LIN {X 0,Y 196.128,Z 397.935,A -85,B 0,C 180,E1 -25531.035,E2 -25531.035} C_VEL
LIN {X 0,Y 198.391,Z 377.082,A -85,B 0,C 180,E1 -25531.639,E2 -25531.639} C_VEL
LIN {X 0,Y 200.245,Z 356.522,A -85,B 0,C 180,E1 -25532.183,E2 -25532.183} C_VEL
LIN {X 0,Y 201.46,Z 342.377,A -85,B 0,C 180,E1 -25532.591,E2 -25532.591} C_VEL
LIN {X 0,Y 197.272,Z 333.633,A -85,B 0,C 180,E1 -25535.814,E2 -25535.814} C_VEL
LIN {X 0,Y 193.686,Z 326.841,A -85,B 0,C 180,E1 -25539.002,E2 -25539.002} C_VEL
LIN {X 0,Y 190.138,Z 320.569,A -85,B 0,C 180,E1 -25542.8,E2 -25542.8} C_VEL
LIN {X 0,Y 187.785,Z 316.689,A -85,B 0,C 180,E1 -25545.92,E2 -25545.92} C_VEL
LIN {X 0,Y 185.741,Z 312.981,A -85,B 0,C 180,E1 -25549.508,E2 -25549.508} C_VEL
LIN {X 0,Y 183.942,Z 310.156,A -85,B 0,C 180,E1 -25554.291,E2 -25554.291} C_VEL
LIN {X 0,Y 183.571,Z 308.41,A -85,B 0,C 180,E1 -25556.708,E2 -25556.708} C_VEL
LIN {X 0,Y 183.342,Z 308.073,A -85,B 0,C 180,E1 -25560,E2 -25560} C_VEL
LIN {X 0,Y 183.573,Z 308.503,A -85,B 0,C 180,E1 -25563.017,E2 -25563.017} C_VEL
LIN {X 0,Y 185.059,Z 312.287,A -85,B 0,C 180,E1 -25568.737,E2 -25568.737} C_VEL
LIN {X 0,Y 185.908,Z 313.347,A -85,B 0,C 180,E1 -25570.493,E2 -25570.493} C_VEL
LIN {X 0,Y 188.57,Z 317.975,A -85,B 0,C 180,E1 -25574.846,E2 -25574.846} C_VEL
LIN {X 0,Y 191.002,Z 322.156,A -85,B 0,C 180,E1 -25577.864,E2 -25577.864} C_VEL
LIN {X 0,Y 194.086,Z 327.519,A -85,B 0,C 180,E1 -25581.021,E2 -25581.021} C_VEL
LIN {X 0,Y 196.464,Z 332.994,A -85,B 0,C 180,E1 -25583.242,E2 -25583.242} C_VEL
LIN {X 0,Y 199.811,Z 341.873,A -85,B 0,C 180,E1 -25586.082,E2 -25586.082} C_VEL
LIN {X 0,Y 201.242,Z 345.874,A -85,B 0,C 180,E1 -25587.202,E2 -25587.202} C_VEL
LIN {X 0,Y 196.159,Z 400.089,A -85,B 0,C 180,E1 -25588.654,E2 -25588.654} C_VEL
LIN {X 0,Y 193.398,Z 415.894,A -85,B 0,C 180,E1 -25589.293,E2 -25589.293} C_VEL
LIN {X 0,Y 189.564,Z 431.114,A -85,B 0,C 180,E1 -25590.2,E2 -25590.2} C_VEL
LIN {X 0,Y 185.029,Z 444.833,A -85,B 0,C 180,E1 -25591.284,E2 -25591.284} C_VEL
LIN {X 0,Y 179.626,Z 458.278,A -85,B 0,C 180,E1 -25592.735,E2 -25592.735} C_VEL
LIN {X 0,Y 173.796,Z 470.579,A -85,B 0,C 180,E1 -25594.481,E2 -25594.481} C_VEL
LIN {X 0,Y 166.767,Z 483.312,A -85,B 0,C 180,E1 -25596.804,E2 -25596.804} C_VEL
LIN {X 0,Y 159.457,Z 494.789,A -85,B 0,C 180,E1 -25599.531,E2 -25599.531} C_VEL
LIN {X 0,Y 152.65,Z 504.457,A -85,B 0,C 180,E1 -25602.556,E2 -25602.556} C_VEL
LIN {X 0,Y 146.078,Z 512.968,A -85,B 0,C 180,E1 -25605.958,E2 -25605.958} C_VEL
LIN {X 0,Y 139.091,Z 521.559,A -85,B 0,C 180,E1 -25610.53,E2 -25610.53} C_VEL
LIN {X 0,Y 132.199,Z 529.29,A -85,B 0,C 180,E1 -25616.069,E2 -25616.069} C_VEL
LIN {X 0,Y 127.359,Z 534.671,A -85,B 0,C 180,E1 -25621.352,E2 -25621.352} C_VEL
LIN {X 0,Y 124.98,Z 536.675,A -85,B 0,C 180,E1 -25623.643,E2 -25623.643} C_VEL
LIN {X 0,Y 119.742,Z 539.495,A -85,B 0,C 180,E1 -25627.37,E2 -25627.37} C_VEL
LIN {X 0,Y 115.773,Z 541.36,A -85,B 0,C 180,E1 -25630.607,E2 -25630.607} C_VEL
LIN {X 0,Y 113.779,Z 542.553,A -85,B 0,C 180,E1 -25633.329,E2 -25633.329} C_VEL
LIN {X 0,Y 113.428,Z 542.855,A -85,B 0,C 180,E1 -25634.29,E2 -25634.29} C_VEL
LIN {X 0,Y 112.457,Z 544.368,A -85,B 0,C 180,E1 -25639.194,E2 -25639.194} C_VEL
LIN {X 0,Y 112.095,Z 545.556,A -85,B 0,C 180,E1 -25646.406,E2 -25646.406} C_VEL
LIN {X 0,Y 112.248,Z 545.716,A -85,B 0,C 180,E1 -25650,E2 -25650} C_VEL
LIN {X 0,Y 112.127,Z 545.085,A -85,B 0,C 180,E1 -25657.201,E2 -25657.201} C_VEL
LIN {X 0,Y 113.102,Z 543.298,A -85,B 0,C 180,E1 -25664.392,E2 -25664.392} C_VEL
LIN {X 0,Y 115.541,Z 540.339,A -85,B 0,C 180,E1 -25671.405,E2 -25671.405} C_VEL
LIN {X 0,Y 119.379,Z 536.141,A -85,B 0,C 180,E1 -25678.097,E2 -25678.097} C_VEL
LIN {X 0,Y 124.755,Z 530.598,A -85,B 0,C 180,E1 -25684.286,E2 -25684.286} C_VEL
LIN {X 0,Y 131.504,Z 523.564,A -85,B 0,C 180,E1 -25689.889,E2 -25689.889} C_VEL
LIN {X 0,Y 138.144,Z 515.994,A -85,B 0,C 180,E1 -25694.427,E2 -25694.427} C_VEL
LIN {X 0,Y 145.607,Z 506.981,A -85,B 0,C 180,E1 -25698.428,E2 -25698.428} C_VEL
LIN {X 0,Y 153.787,Z 496.099,A -85,B 0,C 180,E1 -25702.027,E2 -25702.027} C_VEL
LIN {X 0,Y 161.311,Z 484.904,A -85,B 0,C 180,E1 -25704.774,E2 -25704.774} C_VEL
LIN {X 0,Y 168.603,Z 472.403,A -85,B 0,C 180,E1 -25707.128,E2 -25707.128} C_VEL
LIN {X 0,Y 175.176,Z 459.138,A -85,B 0,C 180,E1 -25709.041,E2 -25709.041} C_VEL
LIN {X 0,Y 180.723,Z 445.878,A -85,B 0,C 180,E1 -25710.471,E2 -25710.471} C_VEL
LIN {X 0,Y 185.34,Z 432.494,A -85,B 0,C 180,E1 -25711.551,E2 -25711.551} C_VEL
LIN {X 0,Y 189.296,Z 417.833,A -85,B 0,C 180,E1 -25712.422,E2 -25712.422} C_VEL
LIN {X 0,Y 192.258,Z 402.311,A -85,B 0,C 180,E1 -25713.067,E2 -25713.067} C_VEL
LIN {X 0,Y 194.771,Z 378.935,A -85,B 0,C 180,E1 -25713.717,E2 -25713.717} C_VEL
LIN {X 0,Y 197.573,Z 348.8,A -85,B 0,C 180,E1 -25714.503,E2 -25714.503} C_VEL
LIN {X 0,Y 194.226,Z 339.095,A -85,B 0,C 180,E1 -25717.53,E2 -25717.53} C_VEL
LIN {X 0,Y 192.008,Z 333.701,A -85,B 0,C 180,E1 -25719.727,E2 -25719.727} C_VEL
LIN {X 0,Y 188.543,Z 327.214,A -85,B 0,C 180,E1 -25723.586,E2 -25723.586} C_VEL
LIN {X 0,Y 186.245,Z 323.237,A -85,B 0,C 180,E1 -25726.776,E2 -25726.776} C_VEL
LIN {X 0,Y 184.286,Z 319.627,A -85,B 0,C 180,E1 -25730.396,E2 -25730.396} C_VEL
LIN {X 0,Y 182.581,Z 316.368,A -85,B 0,C 180,E1 -25735.585,E2 -25735.585} C_VEL
LIN {X 0,Y 182.365,Z 315.273,A -85,B 0,C 180,E1 -25737.239,E2 -25737.239} C_VEL
LIN {X 0,Y 182.148,Z 315.035,A -85,B 0,C 180,E1 -25740,E2 -25740} C_VEL
LIN {X 0,Y 182.427,Z 315.532,A -85,B 0,C 180,E1 -25743.728,E2 -25743.728} C_VEL
LIN {X 0,Y 183.832,Z 319.146,A -85,B 0,C 180,E1 -25749.074,E2 -25749.074} C_VEL
LIN {X 0,Y 184.588,Z 320.208,A -85,B 0,C 180,E1 -25750.697,E2 -25750.697} C_VEL
LIN {X 0,Y 186.924,Z 324.488,A -85,B 0,C 180,E1 -25754.702,E2 -25754.702} C_VEL
LIN {X 0,Y 189.274,Z 328.678,A -85,B 0,C 180,E1 -25757.764,E2 -25757.764} C_VEL
LIN {X 0,Y 191.987,Z 333.709,A -85,B 0,C 180,E1 -25760.701,E2 -25760.701} C_VEL
LIN {X 0,Y 195.196,Z 340.186,A -85,B 0,C 180,E1 -25763.683,E2 -25763.683} C_VEL
LIN {X 0,Y 197.771,Z 345.762,A -85,B 0,C 180,E1 -25765.81,E2 -25765.81} C_VEL
LIN {X 0,Y 193.113,Z 394.413,A -85,B 0,C 180,E1 -25767.114,E2 -25767.114} C_VEL
LIN {X 0,Y 190.393,Z 410.31,A -85,B 0,C 180,E1 -25767.78,E2 -25767.78} C_VEL
LIN {X 0,Y 186.718,Z 425.002,A -85,B 0,C 180,E1 -25768.663,E2 -25768.663} C_VEL
LIN {X 0,Y 182.252,Z 438.791,A -85,B 0,C 180,E1 -25769.816,E2 -25769.816} C_VEL
LIN {X 0,Y 177.003,Z 452.127,A -85,B 0,C 180,E1 -25771.323,E2 -25771.323} C_VEL
LIN {X 0,Y 171.009,Z 464.77,A -85,B 0,C 180,E1 -25773.14,E2 -25773.14} C_VEL
LIN {X 0,Y 164.504,Z 476.331,A -85,B 0,C 180,E1 -25775.21,E2 -25775.21} C_VEL
LIN {X 0,Y 157.683,Z 487.067,A -85,B 0,C 180,E1 -25777.711,E2 -25777.711} C_VEL
LIN {X 0,Y 150.546,Z 496.993,A -85,B 0,C 180,E1 -25780.66,E2 -25780.66} C_VEL
LIN {X 0,Y 143.003,Z 506.676,A -85,B 0,C 180,E1 -25784.553,E2 -25784.553} C_VEL
LIN {X 0,Y 135.891,Z 514.75,A -85,B 0,C 180,E1 -25788.747,E2 -25788.747} C_VEL
LIN {X 0,Y 129.57,Z 521.41,A -85,B 0,C 180,E1 -25793.37,E2 -25793.37} C_VEL
LIN {X 0,Y 123.476,Z 527.564,A -85,B 0,C 180,E1 -25799.186,E2 -25799.186} C_VEL
LIN {X 0,Y 118.71,Z 532.307,A -85,B 0,C 180,E1 -25805.518,E2 -25805.518} C_VEL
LIN {X 0,Y 115.253,Z 535.773,A -85,B 0,C 180,E1 -25812.249,E2 -25812.249} C_VEL
LIN {X 0,Y 113.198,Z 538.054,A -85,B 0,C 180,E1 -25819.266,E2 -25819.266} C_VEL
LIN {X 0,Y 112.353,Z 539.21,A -85,B 0,C 180,E1 -25826.414,E2 -25826.414} C_VEL
LIN {X 0,Y 112.335,Z 539.362,A -85,B 0,C 180,E1 -25830,E2 -25830} C_VEL
LIN {X 0,Y 112.624,Z 538.802,A -85,B 0,C 180,E1 -25837.169,E2 -25837.169} C_VEL
LIN {X 0,Y 114.05,Z 537.13,A -85,B 0,C 180,E1 -25844.269,E2 -25844.269} C_VEL
LIN {X 0,Y 116.718,Z 534.305,A -85,B 0,C 180,E1 -25851.178,E2 -25851.178} C_VEL
LIN {X 0,Y 120.946,Z 530.247,A -85,B 0,C 180,E1 -25857.701,E2 -25857.701} C_VEL
LIN {X 0,Y 126.368,Z 524.865,A -85,B 0,C 180,E1 -25863.789,E2 -25863.789} C_VEL
LIN {X 0,Y 133.011,Z 517.999,A -85,B 0,C 180,E1 -25869.349,E2 -25869.349} C_VEL
LIN {X 0,Y 140.769,Z 509.421,A -85,B 0,C 180,E1 -25874.342,E2 -25874.342} C_VEL
LIN {X 0,Y 147.586,Z 501.119,A -85,B 0,C 180,E1 -25878.012,E2 -25878.012} C_VEL
LIN {X 0,Y 155.159,Z 491.003,A -85,B 0,C 180,E1 -25881.382,E2 -25881.382} C_VEL
LIN {X 0,Y 162.498,Z 479.953,A -85,B 0,C 180,E1 -25884.185,E2 -25884.185} C_VEL
LIN {X 0,Y 169.582,Z 467.84,A -85,B 0,C 180,E1 -25886.514,E2 -25886.514} C_VEL
LIN {X 0,Y 175.733,Z 455.423,A -85,B 0,C 180,E1 -25888.398,E2 -25888.398} C_VEL
LIN {X 0,Y 180.809,Z 443.245,A -85,B 0,C 180,E1 -25889.863,E2 -25889.863} C_VEL
LIN {X 0,Y 185.929,Z 428.329,A -85,B 0,C 180,E1 -25891.217,E2 -25891.217} C_VEL
LIN {X 0,Y 189.927,Z 413.246,A -85,B 0,C 180,E1 -25892.202,E2 -25892.202} C_VEL
LIN {X 0,Y 192.784,Z 398.214,A -85,B 0,C 180,E1 -25892.874,E2 -25892.874} C_VEL
LIN {X 0,Y 195.151,Z 377.016,A -85,B 0,C 180,E1 -25893.474,E2 -25893.474} C_VEL
LIN {X 0,Y 196.842,Z 358.585,A -85,B 0,C 180,E1 -25893.969,E2 -25893.969} C_VEL
LIN {X 0,Y 197.973,Z 345.87,A -85,B 0,C 180,E1 -25894.332,E2 -25894.332} C_VEL
LIN {X 0,Y 194.145,Z 337.65,A -85,B 0,C 180,E1 -25897.59,E2 -25897.59} C_VEL
LIN {X 0,Y 190.481,Z 330.553,A -85,B 0,C 180,E1 -25901.27,E2 -25901.27} C_VEL
LIN {X 0,Y 188.099,Z 326.329,A -85,B 0,C 180,E1 -25904.144,E2 -25904.144} C_VEL
LIN {X 0,Y 186.4,Z 323.297,A -85,B 0,C 180,E1 -25906.619,E2 -25906.619} C_VEL
LIN {X 0,Y 184.406,Z 319.665,A -85,B 0,C 180,E1 -25910.402,E2 -25910.402} C_VEL
LIN {X 0,Y 182.733,Z 316.096,A -85,B 0,C 180,E1 -25916.141,E2 -25916.141} C_VEL
LIN {X 0,Y 182.63,Z 315.373,A -85,B 0,C 180,E1 -25917.243,E2 -25917.243} C_VEL
LIN {X 0,Y 182.477,Z 315.121,A -85,B 0,C 180,E1 -25920,E2 -25920} C_VEL
LIN {X 0,Y 182.67,Z 315.579,A -85,B 0,C 180,E1 -25922.825,E2 -25922.825} C_VEL
LIN {X 0,Y 184.076,Z 319.279,A -85,B 0,C 180,E1 -25928.508,E2 -25928.508} C_VEL
LIN {X 0,Y 184.77,Z 320.244,A -85,B 0,C 180,E1 -25930.028,E2 -25930.028} C_VEL
LIN {X 0,Y 187.212,Z 324.704,A -85,B 0,C 180,E1 -25934.262,E2 -25934.262} C_VEL
LIN {X 0,Y 189.498,Z 328.843,A -85,B 0,C 180,E1 -25937.259,E2 -25937.259} C_VEL
LIN {X 0,Y 192.256,Z 333.937,A -85,B 0,C 180,E1 -25940.251,E2 -25940.251} C_VEL
LIN {X 0,Y 194.505,Z 339.504,A -85,B 0,C 180,E1 -25942.49,E2 -25942.49} C_VEL
LIN {X 0,Y 197.731,Z 348.761,A -85,B 0,C 180,E1 -25945.407,E2 -25945.407} C_VEL
LIN {X 0,Y 197.495,Z 352.481,A -85,B 0,C 180,E1 -25945.57,E2 -25945.57} C_VEL
LIN {X 0,Y 192.822,Z 400.102,A -85,B 0,C 180,E1 -25946.807,E2 -25946.807} C_VEL
LIN {X 0,Y 190.035,Z 415.703,A -85,B 0,C 180,E1 -25947.432,E2 -25947.432} C_VEL
LIN {X 0,Y 186.098,Z 430.92,A -85,B 0,C 180,E1 -25948.312,E2 -25948.312} C_VEL
LIN {X 0,Y 181.442,Z 444.638,A -85,B 0,C 180,E1 -25949.367,E2 -25949.367} C_VEL
LIN {X 0,Y 175.887,Z 458.082,A -85,B 0,C 180,E1 -25950.788,E2 -25950.788} C_VEL
LIN {X 0,Y 169.464,Z 471.172,A -85,B 0,C 180,E1 -25952.624,E2 -25952.624} C_VEL
LIN {X 0,Y 161.953,Z 484.186,A -85,B 0,C 180,E1 -25955.008,E2 -25955.008} C_VEL
LIN {X 0,Y 153.794,Z 496.35,A -85,B 0,C 180,E1 -25957.977,E2 -25957.977} C_VEL
LIN {X 0,Y 145.615,Z 507.182,A -85,B 0,C 180,E1 -25961.576,E2 -25961.576} C_VEL
LIN {X 0,Y 138.219,Z 516.099,A -85,B 0,C 180,E1 -25965.541,E2 -25965.541} C_VEL
LIN {X 0,Y 131.509,Z 523.718,A -85,B 0,C 180,E1 -25970.113,E2 -25970.113} C_VEL
LIN {X 0,Y 124.778,Z 530.716,A -85,B 0,C 180,E1 -25975.721,E2 -25975.721} C_VEL
LIN {X 0,Y 119.282,Z 536.375,A -85,B 0,C 180,E1 -25982.102,E2 -25982.102} C_VEL
LIN {X 0,Y 115.57,Z 540.407,A -85,B 0,C 180,E1 -25988.601,E2 -25988.601} C_VEL
LIN {X 0,Y 113.428,Z 542.855,A -85,B 0,C 180,E1 -25994.29,E2 -25994.29} C_VEL
LIN {X 0,Y 112.204,Z 543.852,A -85,B 0,C 180,E1 -25997.178,E2 -25997.178} C_VEL
LIN {X 0,Y 109.003,Z 544.995,A -85,B 0,C 180,E1 -26001.986,E2 -26001.986} C_VEL
LIN {X 0,Y 105.6,Z 545.541,A -85,B 0,C 180,E1 -26008.126,E2 -26008.126} C_VEL
LIN {X 0,Y 105.138,Z 545.503,A -85,B 0,C 180,E1 -26010.282,E2 -26010.282} C_VEL
LIN {X 0,Y 105.053,Z 544.883,A -85,B 0,C 180,E1 -26017.689,E2 -26017.689} C_VEL
LIN {X 0,Y 106.184,Z 543.095,A -85,B 0,C 180,E1 -26025.352,E2 -26025.352} C_VEL
LIN {X 0,Y 108.884,Z 540.135,A -85,B 0,C 180,E1 -26032.785,E2 -26032.785} C_VEL
LIN {X 0,Y 113.108,Z 535.937,A -85,B 0,C 180,E1 -26039.806,E2 -26039.806} C_VEL
LIN {X 0,Y 118.895,Z 530.394,A -85,B 0,C 180,E1 -26046.235,E2 -26046.235} C_VEL
LIN {X 0,Y 126.06,Z 523.358,A -85,B 0,C 180,E1 -26051.99,E2 -26051.99} C_VEL
LIN {X 0,Y 133.554,Z 515.296,A -85,B 0,C 180,E1 -26056.836,E2 -26056.836} C_VEL
LIN {X 0,Y 140.964,Z 506.777,A -85,B 0,C 180,E1 -26060.602,E2 -26060.602} C_VEL
LIN {X 0,Y 149.493,Z 495.894,A -85,B 0,C 180,E1 -26064.188,E2 -26064.188} C_VEL
LIN {X 0,Y 157.313,Z 484.7,A -85,B 0,C 180,E1 -26066.892,E2 -26066.892} C_VEL
LIN {X 0,Y 165.105,Z 471.735,A -85,B 0,C 180,E1 -26069.283,E2 -26069.283} C_VEL
LIN {X 0,Y 171.628,Z 458.933,A -85,B 0,C 180,E1 -26071.077,E2 -26071.077} C_VEL
LIN {X 0,Y 177.327,Z 445.672,A -85,B 0,C 180,E1 -26072.47,E2 -26072.47} C_VEL
LIN {X 0,Y 182.069,Z 432.286,A -85,B 0,C 180,E1 -26073.513,E2 -26073.513} C_VEL
LIN {X 0,Y 186.12,Z 417.623,A -85,B 0,C 180,E1 -26074.358,E2 -26074.358} C_VEL
LIN {X 0,Y 189.102,Z 402.418,A -85,B 0,C 180,E1 -26074.97,E2 -26074.97} C_VEL
LIN {X 0,Y 191.639,Z 379.78,A -85,B 0,C 180,E1 -26075.587,E2 -26075.587} C_VEL
LIN {X 0,Y 194.302,Z 351.818,A -85,B 0,C 180,E1 -26076.313,E2 -26076.313} C_VEL
LIN {X 0,Y 191.403,Z 343.066,A -85,B 0,C 180,E1 -26079.234,E2 -26079.234} C_VEL
LIN {X 0,Y 189.685,Z 339.028,A -85,B 0,C 180,E1 -26081.083,E2 -26081.083} C_VEL
LIN {X 0,Y 186.8,Z 333.397,A -85,B 0,C 180,E1 -26084.591,E2 -26084.591} C_VEL
LIN {X 0,Y 184.86,Z 329.819,A -85,B 0,C 180,E1 -26087.513,E2 -26087.513} C_VEL
LIN {X 0,Y 183.131,Z 326.461,A -85,B 0,C 180,E1 -26090.961,E2 -26090.961} C_VEL
LIN {X 0,Y 181.541,Z 322.805,A -85,B 0,C 180,E1 -26096.671,E2 -26096.671} C_VEL
LIN {X 0,Y 181.425,Z 322.252,A -85,B 0,C 180,E1 -26097.78,E2 -26097.78} C_VEL
LIN {X 0,Y 181.437,Z 322.287,A -85,B 0,C 180,E1 -26102.776,E2 -26102.776} C_VEL
LIN {X 0,Y 183.089,Z 326.414,A -85,B 0,C 180,E1 -26109.389,E2 -26109.389} C_VEL
LIN {X 0,Y 185.397,Z 330.78,A -85,B 0,C 180,E1 -26113.802,E2 -26113.802} C_VEL
LIN {X 0,Y 187.834,Z 335.446,A -85,B 0,C 180,E1 -26117.207,E2 -26117.207} C_VEL
LIN {X 0,Y 190.678,Z 341.118,A -85,B 0,C 180,E1 -26120.426,E2 -26120.426} C_VEL
LIN {X 0,Y 193.81,Z 347.891,A -85,B 0,C 180,E1 -26123.441,E2 -26123.441} C_VEL
LIN {X 0,Y 194.453,Z 349.345,A -85,B 0,C 180,E1 -26124.009,E2 -26124.009} C_VEL
LIN {X 0,Y 189.897,Z 395.315,A -85,B 0,C 180,E1 -26125.238,E2 -26125.238} C_VEL
LIN {X 0,Y 187.193,Z 410.521,A -85,B 0,C 180,E1 -26125.859,E2 -26125.859} C_VEL
LIN {X 0,Y 183.429,Z 425.211,A -85,B 0,C 180,E1 -26126.723,E2 -26126.723} C_VEL
LIN {X 0,Y 178.824,Z 438.999,A -85,B 0,C 180,E1 -26127.84,E2 -26127.84} C_VEL
LIN {X 0,Y 173.211,Z 452.802,A -85,B 0,C 180,E1 -26129.373,E2 -26129.373} C_VEL
LIN {X 0,Y 166.561,Z 466.262,A -85,B 0,C 180,E1 -26131.304,E2 -26131.304} C_VEL
LIN {X 0,Y 159.211,Z 478.664,A -85,B 0,C 180,E1 -26133.574,E2 -26133.574} C_VEL
LIN {X 0,Y 152.16,Z 489.045,A -85,B 0,C 180,E1 -26136.072,E2 -26136.072} C_VEL
LIN {X 0,Y 144.086,Z 499.542,A -85,B 0,C 180,E1 -26139.353,E2 -26139.353} C_VEL
LIN {X 0,Y 136.978,Z 508.102,A -85,B 0,C 180,E1 -26143.02,E2 -26143.02} C_VEL
LIN {X 0,Y 129.609,Z 515.954,A -85,B 0,C 180,E1 -26147.329,E2 -26147.329} C_VEL
LIN {X 0,Y 122.173,Z 523.278,A -85,B 0,C 180,E1 -26152.843,E2 -26152.843} C_VEL
LIN {X 0,Y 115.975,Z 529.079,A -85,B 0,C 180,E1 -26158.997,E2 -26158.997} C_VEL
LIN {X 0,Y 112.273,Z 532.509,A -85,B 0,C 180,E1 -26164.013,E2 -26164.013} C_VEL
LIN {X 0,Y 108.478,Z 535.975,A -85,B 0,C 180,E1 -26171.099,E2 -26171.099} C_VEL
LIN {X 0,Y 106.212,Z 538.256,A -85,B 0,C 180,E1 -26178.55,E2 -26178.55} C_VEL
LIN {X 0,Y 105.265,Z 539.411,A -85,B 0,C 180,E1 -26186.172,E2 -26186.172} C_VEL
LIN {X 0,Y 105.237,Z 539.563,A -85,B 0,C 180,E1 -26190,E2 -26190} C_VEL
LIN {X 0,Y 105.592,Z 539.003,A -85,B 0,C 180,E1 -26197.649,E2 -26197.649} C_VEL
LIN {X 0,Y 107.157,Z 537.331,A -85,B 0,C 180,E1 -26205.209,E2 -26205.209} C_VEL
LIN {X 0,Y 110.094,Z 534.506,A -85,B 0,C 180,E1 -26212.52,E2 -26212.52} C_VEL
LIN {X 0,Y 114.654,Z 530.449,A -85,B 0,C 180,E1 -26219.365,E2 -26219.365} C_VEL
LIN {X 0,Y 120.496,Z 525.066,A -85,B 0,C 180,E1 -26225.679,E2 -26225.679} C_VEL
LIN {X 0,Y 127.58,Z 518.199,A -85,B 0,C 180,E1 -26231.378,E2 -26231.378} C_VEL
LIN {X 0,Y 134.663,Z 510.816,A -85,B 0,C 180,E1 -26235.856,E2 -26235.856} C_VEL
LIN {X 0,Y 141.344,Z 503.199,A -85,B 0,C 180,E1 -26239.355,E2 -26239.355} C_VEL
LIN {X 0,Y 147.146,Z 496.054,A -85,B 0,C 180,E1 -26242.004,E2 -26242.004} C_VEL
LIN {X 0,Y 154.657,Z 485.912,A -85,B 0,C 180,E1 -26244.879,E2 -26244.879} C_VEL
LIN {X 0,Y 161.081,Z 475.963,A -85,B 0,C 180,E1 -26247.125,E2 -26247.125} C_VEL
LIN {X 0,Y 168.494,Z 462.994,A -85,B 0,C 180,E1 -26249.346,E2 -26249.346} C_VEL
LIN {X 0,Y 174.472,Z 450.327,A -85,B 0,C 180,E1 -26251.093,E2 -26251.093} C_VEL
LIN {X 0,Y 180.152,Z 435.959,A -85,B 0,C 180,E1 -26252.559,E2 -26252.559} C_VEL
LIN {X 0,Y 184.773,Z 421.22,A -85,B 0,C 180,E1 -26253.663,E2 -26253.663} C_VEL
LIN {X 0,Y 188.18,Z 406.625,A -85,B 0,C 180,E1 -26254.466,E2 -26254.466} C_VEL
LIN {X 0,Y 190.714,Z 390.557,A -85,B 0,C 180,E1 -26255.032,E2 -26255.032} C_VEL
LIN {X 0,Y 192.711,Z 370.089,A -85,B 0,C 180,E1 -26255.588,E2 -26255.588} C_VEL
LIN {X 0,Y 194.695,Z 349.528,A -85,B 0,C 180,E1 -26256.106,E2 -26256.106} C_VEL
LIN {X 0,Y 191.57,Z 342.573,A -85,B 0,C 180,E1 -26259.041,E2 -26259.041} C_VEL
LIN {X 0,Y 188.427,Z 336.273,A -85,B 0,C 180,E1 -26262.499,E2 -26262.499} C_VEL
LIN {X 0,Y 186.624,Z 332.876,A -85,B 0,C 180,E1 -26264.86,E2 -26264.86} C_VEL
LIN {X 0,Y 185.088,Z 330.002,A -85,B 0,C 180,E1 -26267.249,E2 -26267.249} C_VEL
LIN {X 0,Y 183.297,Z 326.501,A -85,B 0,C 180,E1 -26270.9,E2 -26270.9} C_VEL
LIN {X 0,Y 181.792,Z 322.923,A -85,B 0,C 180,E1 -26276.675,E2 -26276.675} C_VEL
LIN {X 0,Y 181.704,Z 322.347,A -85,B 0,C 180,E1 -26277.783,E2 -26277.783} C_VEL
LIN {X 0,Y 181.645,Z 322.261,A -85,B 0,C 180,E1 -26281.108,E2 -26281.108} C_VEL
LIN {X 0,Y 181.767,Z 322.671,A -85,B 0,C 180,E1 -26282.631,E2 -26282.631} C_VEL
LIN {X 0,Y 183.095,Z 326.274,A -85,B 0,C 180,E1 -26288.276,E2 -26288.276} C_VEL
LIN {X 0,Y 183.692,Z 327.201,A -85,B 0,C 180,E1 -26289.659,E2 -26289.659} C_VEL
LIN {X 0,Y 185.874,Z 331.433,A -85,B 0,C 180,E1 -26293.669,E2 -26293.669} C_VEL
LIN {X 0,Y 187.954,Z 335.392,A -85,B 0,C 180,E1 -26296.565,E2 -26296.565} C_VEL
LIN {X 0,Y 190.76,Z 340.985,A -85,B 0,C 180,E1 -26299.784,E2 -26299.784} C_VEL
LIN {X 0,Y 193.285,Z 348.192,A -85,B 0,C 180,E1 -26302.444,E2 -26302.444} C_VEL
LIN {X 0,Y 194.524,Z 352.047,A -85,B 0,C 180,E1 -26303.652,E2 -26303.652} C_VEL
LIN {X 0,Y 189.706,Z 400.09,A -85,B 0,C 180,E1 -26304.904,E2 -26304.904} C_VEL
LIN {X 0,Y 186.859,Z 415.511,A -85,B 0,C 180,E1 -26305.492,E2 -26305.492} C_VEL
LIN {X 0,Y 182.841,Z 430.726,A -85,B 0,C 180,E1 -26306.355,E2 -26306.355} C_VEL
LIN {X 0,Y 178.066,Z 444.442,A -85,B 0,C 180,E1 -26307.375,E2 -26307.375} C_VEL
LIN {X 0,Y 172.357,Z 457.886,A -85,B 0,C 180,E1 -26308.758,E2 -26308.758} C_VEL
LIN {X 0,Y 166.014,Z 470.454,A -85,B 0,C 180,E1 -26310.474,E2 -26310.474} C_VEL
LIN {X 0,Y 158.644,Z 482.916,A -85,B 0,C 180,E1 -26312.681,E2 -26312.681} C_VEL
LIN {X 0,Y 150.754,Z 494.39,A -85,B 0,C 180,E1 -26315.332,E2 -26315.332} C_VEL
LIN {X 0,Y 143.355,Z 504.057,A -85,B 0,C 180,E1 -26318.336,E2 -26318.336} C_VEL
LIN {X 0,Y 135.263,Z 513.558,A -85,B 0,C 180,E1 -26322.236,E2 -26322.236} C_VEL
LIN {X 0,Y 128.011,Z 521.485,A -85,B 0,C 180,E1 -26326.666,E2 -26326.666} C_VEL
LIN {X 0,Y 120.555,Z 528.886,A -85,B 0,C 180,E1 -26332.258,E2 -26332.258} C_VEL
LIN {X 0,Y 114.462,Z 534.769,A -85,B 0,C 180,E1 -26338.541,E2 -26338.541} C_VEL
LIN {X 0,Y 110.885,Z 538.277,A -85,B 0,C 180,E1 -26343.663,E2 -26343.663} C_VEL
LIN {X 0,Y 107.318,Z 541.822,A -85,B 0,C 180,E1 -26350.887,E2 -26350.887} C_VEL
LIN {X 0,Y 105.463,Z 544.167,A -85,B 0,C 180,E1 -26358.468,E2 -26358.468} C_VEL
LIN {X 0,Y 105.005,Z 545.355,A -85,B 0,C 180,E1 -26366.162,E2 -26366.162} C_VEL
LIN {X 0,Y 105.138,Z 545.503,A -85,B 0,C 180,E1 -26370.282,E2 -26370.282} C_VEL
LIN {X 0,Y 104.271,Z 545.349,A -85,B 0,C 180,E1 -26373.475,E2 -26373.475} C_VEL
LIN {X 0,Y 101.537,Z 544.676,A -85,B 0,C 180,E1 -26378.775,E2 -26378.775} C_VEL
LIN {X 0,Y 99.684,Z 543.768,A -85,B 0,C 180,E1 -26383.182,E2 -26383.182} C_VEL
LIN {X 0,Y 99.396,Z 542.856,A -85,B 0,C 180,E1 -26386.568,E2 -26386.568} C_VEL
LIN {X 0,Y 99.626,Z 542.484,A -85,B 0,C 180,E1 -26387.685,E2 -26387.685} C_VEL
LIN {X 0,Y 102.3,Z 539.932,A -85,B 0,C 180,E1 -26394.343,E2 -26394.343} C_VEL
LIN {X 0,Y 106.942,Z 535.733,A -85,B 0,C 180,E1 -26401.717,E2 -26401.717} C_VEL
LIN {X 0,Y 113.178,Z 530.189,A -85,B 0,C 180,E1 -26408.386,E2 -26408.386} C_VEL
LIN {X 0,Y 120.824,Z 523.154,A -85,B 0,C 180,E1 -26414.266,E2 -26414.266} C_VEL
LIN {X 0,Y 128.167,Z 515.711,A -85,B 0,C 180,E1 -26418.852,E2 -26418.852} C_VEL
LIN {X 0,Y 136.53,Z 506.572,A -85,B 0,C 180,E1 -26422.926,E2 -26422.926} C_VEL
LIN {X 0,Y 145.416,Z 495.689,A -85,B 0,C 180,E1 -26426.478,E2 -26426.478} C_VEL
LIN {X 0,Y 153.539,Z 484.495,A -85,B 0,C 180,E1 -26429.119,E2 -26429.119} C_VEL
LIN {X 0,Y 161.037,Z 472.448,A -85,B 0,C 180,E1 -26431.311,E2 -26431.311} C_VEL
LIN {X 0,Y 168.293,Z 458.726,A -85,B 0,C 180,E1 -26433.203,E2 -26433.203} C_VEL
LIN {X 0,Y 174.154,Z 445.465,A -85,B 0,C 180,E1 -26434.545,E2 -26434.545} C_VEL
LIN {X 0,Y 179.013,Z 432.078,A -85,B 0,C 180,E1 -26435.549,E2 -26435.549} C_VEL
LIN {X 0,Y 183.163,Z 417.413,A -85,B 0,C 180,E1 -26436.358,E2 -26436.358} C_VEL
LIN {X 0,Y 186.243,Z 401.971,A -85,B 0,C 180,E1 -26436.96,E2 -26436.96} C_VEL
LIN {X 0,Y 188.911,Z 378.6,A -85,B 0,C 180,E1 -26437.572,E2 -26437.572} C_VEL
LIN {X 0,Y 191.202,Z 354.974,A -85,B 0,C 180,E1 -26438.193,E2 -26438.193} C_VEL
LIN {X 0,Y 189.01,Z 347.982,A -85,B 0,C 180,E1 -26440.661,E2 -26440.661} C_VEL
LIN {X 0,Y 187.355,Z 344.152,A -85,B 0,C 180,E1 -26442.607,E2 -26442.607} C_VEL
LIN {X 0,Y 185.056,Z 339.435,A -85,B 0,C 180,E1 -26445.709,E2 -26445.709} C_VEL
LIN {X 0,Y 183.544,Z 336.474,A -85,B 0,C 180,E1 -26448.193,E2 -26448.193} C_VEL
LIN {X 0,Y 182.054,Z 333.339,A -85,B 0,C 180,E1 -26451.397,E2 -26451.397} C_VEL
LIN {X 0,Y 180.621,Z 329.781,A -85,B 0,C 180,E1 -26457.003,E2 -26457.003} C_VEL
LIN {X 0,Y 180.56,Z 329.306,A -85,B 0,C 180,E1 -26457.77,E2 -26457.77} C_VEL
LIN {X 0,Y 180.507,Z 329.298,A -85,B 0,C 180,E1 -26462.232,E2 -26462.232} C_VEL
LIN {X 0,Y 180.645,Z 329.965,A -85,B 0,C 180,E1 -26463.695,E2 -26463.695} C_VEL
LIN {X 0,Y 181.985,Z 333.268,A -85,B 0,C 180,E1 -26468.887,E2 -26468.887} C_VEL
LIN {X 0,Y 184.035,Z 337.372,A -85,B 0,C 180,E1 -26473.103,E2 -26473.103} C_VEL
LIN {X 0,Y 186.261,Z 341.887,A -85,B 0,C 180,E1 -26476.439,E2 -26476.439} C_VEL
LIN {X 0,Y 189.169,Z 348.042,A -85,B 0,C 180,E1 -26479.924,E2 -26479.924} C_VEL
LIN {X 0,Y 191.366,Z 353.104,A -85,B 0,C 180,E1 -26482.189,E2 -26482.189} C_VEL
LIN {X 0,Y 186.918,Z 395.964,A -85,B 0,C 180,E1 -26483.29,E2 -26483.29} C_VEL
LIN {X 0,Y 184.028,Z 411.498,A -85,B 0,C 180,E1 -26483.915,E2 -26483.915} C_VEL
LIN {X 0,Y 179.989,Z 426.568,A -85,B 0,C 180,E1 -26484.795,E2 -26484.795} C_VEL
LIN {X 0,Y 174.908,Z 441.061,A -85,B 0,C 180,E1 -26485.969,E2 -26485.969} C_VEL
LIN {X 0,Y 168.893,Z 455.011,A -85,B 0,C 180,E1 -26487.532,E2 -26487.532} C_VEL
LIN {X 0,Y 162.283,Z 467.704,A -85,B 0,C 180,E1 -26489.363,E2 -26489.363} C_VEL
LIN {X 0,Y 154.717,Z 479.902,A -85,B 0,C 180,E1 -26491.603,E2 -26491.603} C_VEL
LIN {X 0,Y 146.771,Z 491.014,A -85,B 0,C 180,E1 -26494.312,E2 -26494.312} C_VEL
LIN {X 0,Y 138.234,Z 501.537,A -85,B 0,C 180,E1 -26497.774,E2 -26497.774} C_VEL
LIN {X 0,Y 131.057,Z 509.529,A -85,B 0,C 180,E1 -26501.345,E2 -26501.345} C_VEL
LIN {X 0,Y 123.425,Z 517.157,A -85,B 0,C 180,E1 -26505.772,E2 -26505.772} C_VEL
LIN {X 0,Y 116.562,Z 523.481,A -85,B 0,C 180,E1 -26510.723,E2 -26510.723} C_VEL
LIN {X 0,Y 109.918,Z 529.282,A -85,B 0,C 180,E1 -26517.08,E2 -26517.08} C_VEL
LIN {X 0,Y 105.908,Z 532.711,A -85,B 0,C 180,E1 -26522.322,E2 -26522.322} C_VEL
LIN {X 0,Y 101.76,Z 536.178,A -85,B 0,C 180,E1 -26529.799,E2 -26529.799} C_VEL
LIN {X 0,Y 99.257,Z 538.457,A -85,B 0,C 180,E1 -26537.736,E2 -26537.736} C_VEL
LIN {X 0,Y 98.189,Z 539.612,A -85,B 0,C 180,E1 -26545.896,E2 -26545.896} C_VEL
LIN {X 0,Y 98.151,Z 539.763,A -85,B 0,C 180,E1 -26550,E2 -26550} C_VEL
LIN {X 0,Y 98.553,Z 539.203,A -85,B 0,C 180,E1 -26558.199,E2 -26558.199} C_VEL
LIN {X 0,Y 100.306,Z 537.532,A -85,B 0,C 180,E1 -26566.275,E2 -26566.275} C_VEL
LIN {X 0,Y 103.54,Z 534.707,A -85,B 0,C 180,E1 -26574.032,E2 -26574.032} C_VEL
LIN {X 0,Y 108.475,Z 530.65,A -85,B 0,C 180,E1 -26581.218,E2 -26581.218} C_VEL
LIN {X 0,Y 114.773,Z 525.266,A -85,B 0,C 180,E1 -26587.758,E2 -26587.758} C_VEL
LIN {X 0,Y 122.32,Z 518.399,A -85,B 0,C 180,E1 -26593.587,E2 -26593.587} C_VEL
LIN {X 0,Y 129.812,Z 511.016,A -85,B 0,C 180,E1 -26598.108,E2 -26598.108} C_VEL
LIN {X 0,Y 137.574,Z 502.496,A -85,B 0,C 180,E1 -26602.012,E2 -26602.012} C_VEL
LIN {X 0,Y 145.405,Z 493.02,A -85,B 0,C 180,E1 -26605.251,E2 -26605.251} C_VEL
LIN {X 0,Y 153.266,Z 482.292,A -85,B 0,C 180,E1 -26608.027,E2 -26608.027} C_VEL
LIN {X 0,Y 160.775,Z 470.574,A -85,B 0,C 180,E1 -26610.317,E2 -26610.317} C_VEL
LIN {X 0,Y 167.736,Z 457.801,A -85,B 0,C 180,E1 -26612.251,E2 -26612.251} C_VEL
LIN {X 0,Y 173.407,Z 445.396,A -85,B 0,C 180,E1 -26613.725,E2 -26613.725} C_VEL
LIN {X 0,Y 178.447,Z 432.097,A -85,B 0,C 180,E1 -26614.933,E2 -26614.933} C_VEL
LIN {X 0,Y 182.823,Z 417.431,A -85,B 0,C 180,E1 -26615.918,E2 -26615.918} C_VEL
LIN {X 0,Y 186.146,Z 402.287,A -85,B 0,C 180,E1 -26616.622,E2 -26616.622} C_VEL
LIN {X 0,Y 188.375,Z 386.071,A -85,B 0,C 180,E1 -26617.109,E2 -26617.109} C_VEL
LIN {X 0,Y 191.596,Z 353.22,A -85,B 0,C 180,E1 -26617.946,E2 -26617.946} C_VEL
LIN {X 0,Y 188.628,Z 346.504,A -85,B 0,C 180,E1 -26621.079,E2 -26621.079} C_VEL
LIN {X 0,Y 185.733,Z 340.396,A -85,B 0,C 180,E1 -26624.786,E2 -26624.786} C_VEL
LIN {X 0,Y 183.817,Z 336.711,A -85,B 0,C 180,E1 -26627.861,E2 -26627.861} C_VEL
LIN {X 0,Y 182.2,Z 333.363,A -85,B 0,C 180,E1 -26631.404,E2 -26631.404} C_VEL
LIN {X 0,Y 180.867,Z 329.751,A -85,B 0,C 180,E1 -26637.216,E2 -26637.216} C_VEL
LIN {X 0,Y 180.759,Z 329.298,A -85,B 0,C 180,E1 -26638.886,E2 -26638.886} C_VEL
LIN {X 0,Y 180.851,Z 329.5,A -85,B 0,C 180,E1 -26642.088,E2 -26642.088} C_VEL
LIN {X 0,Y 182.118,Z 333.265,A -85,B 0,C 180,E1 -26648.041,E2 -26648.041} C_VEL
LIN {X 0,Y 182.612,Z 334.197,A -85,B 0,C 180,E1 -26649.274,E2 -26649.274} C_VEL
LIN {X 0,Y 184.478,Z 337.976,A -85,B 0,C 180,E1 -26652.933,E2 -26652.933} C_VEL
LIN {X 0,Y 186.573,Z 342.194,A -85,B 0,C 180,E1 -26656.038,E2 -26656.038} C_VEL
LIN {X 0,Y 188.873,Z 347.147,A -85,B 0,C 180,E1 -26658.86,E2 -26658.86} C_VEL
LIN {X 0,Y 191.117,Z 354.155,A -85,B 0,C 180,E1 -26661.434,E2 -26661.434} C_VEL
LIN {X 0,Y 191.475,Z 355.303,A -85,B 0,C 180,E1 -26661.816,E2 -26661.816} C_VEL
LIN {X 0,Y 186.823,Z 399.988,A -85,B 0,C 180,E1 -26662.939,E2 -26662.939} C_VEL
LIN {X 0,Y 183.905,Z 415.319,A -85,B 0,C 180,E1 -26663.488,E2 -26663.488} C_VEL
LIN {X 0,Y 179.801,Z 430.532,A -85,B 0,C 180,E1 -26664.327,E2 -26664.327} C_VEL
LIN {X 0,Y 174.915,Z 444.247,A -85,B 0,C 180,E1 -26665.309,E2 -26665.309} C_VEL
LIN {X 0,Y 169.037,Z 457.689,A -85,B 0,C 180,E1 -26666.635,E2 -26666.635} C_VEL
LIN {X 0,Y 162.102,Z 471.002,A -85,B 0,C 180,E1 -26668.414,E2 -26668.414} C_VEL
LIN {X 0,Y 154.228,Z 483.79,A -85,B 0,C 180,E1 -26670.673,E2 -26670.673} C_VEL
LIN {X 0,Y 145.424,Z 495.951,A -85,B 0,C 180,E1 -26673.526,E2 -26673.526} C_VEL
LIN {X 0,Y 136.54,Z 506.782,A -85,B 0,C 180,E1 -26677.079,E2 -26677.079} C_VEL
LIN {X 0,Y 128.246,Z 515.822,A -85,B 0,C 180,E1 -26681.118,E2 -26681.118} C_VEL
LIN {X 0,Y 120.832,Z 523.315,A -85,B 0,C 180,E1 -26685.738,E2 -26685.738} C_VEL
LIN {X 0,Y 113.198,Z 530.312,A -85,B 0,C 180,E1 -26691.622,E2 -26691.622} C_VEL
LIN {X 0,Y 106.992,Z 535.825,A -85,B 0,C 180,E1 -26698.299,E2 -26698.299} C_VEL
LIN {X 0,Y 102.347,Z 540.002,A -85,B 0,C 180,E1 -26705.67,E2 -26705.67} C_VEL
LIN {X 0,Y 99.299,Z 542.939,A -85,B 0,C 180,E1 -26713.555,E2 -26713.555} C_VEL
LIN {X 0,Y 98.005,Z 544.702,A -85,B 0,C 180,E1 -26721.754,E2 -26721.754} C_VEL
LIN {X 0,Y 98.066,Z 545.313,A -85,B 0,C 180,E1 -26730.056,E2 -26730.056} C_VEL
LIN {X 0,Y 98.004,Z 544.682,A -85,B 0,C 180,E1 -26738.246,E2 -26738.246} C_VEL
LIN {X 0,Y 99.285,Z 542.891,A -85,B 0,C 180,E1 -26746.448,E2 -26746.448} C_VEL
LIN {X 0,Y 99.626,Z 542.484,A -85,B 0,C 180,E1 -26747.685,E2 -26747.685} C_VEL
LIN {X 0,Y 100.081,Z 541.4,A -85,B 0,C 180,E1 -26751.002,E2 -26751.002} C_VEL
LIN {X 0,Y 99.719,Z 539.205,A -85,B 0,C 180,E1 -26756.555,E2 -26756.555} C_VEL
LIN {X 0,Y 99.925,Z 537.139,A -85,B 0,C 180,E1 -26760.968,E2 -26760.968} C_VEL
LIN {X 0,Y 101.204,Z 535.356,A -85,B 0,C 180,E1 -26764.1,E2 -26764.1} C_VEL
LIN {X 0,Y 101.943,Z 534.69,A -85,B 0,C 180,E1 -26765.066,E2 -26765.066} C_VEL
LIN {X 0,Y 109.567,Z 528.356,A -85,B 0,C 180,E1 -26772.337,E2 -26772.337} C_VEL
LIN {X 0,Y 117.928,Z 520.915,A -85,B 0,C 180,E1 -26778.153,E2 -26778.153} C_VEL
LIN {X 0,Y 126.047,Z 512.959,A -85,B 0,C 180,E1 -26782.61,E2 -26782.61} C_VEL
LIN {X 0,Y 134.938,Z 503.421,A -85,B 0,C 180,E1 -26786.44,E2 -26786.44} C_VEL
LIN {X 0,Y 142.959,Z 493.706,A -85,B 0,C 180,E1 -26789.35,E2 -26789.35} C_VEL
LIN {X 0,Y 151.426,Z 482.183,A -85,B 0,C 180,E1 -26791.862,E2 -26791.862} C_VEL
LIN {X 0,Y 159.311,Z 469.484,A -85,B 0,C 180,E1 -26794.004,E2 -26794.004} C_VEL
LIN {X 0,Y 165.945,Z 456.976,A -85,B 0,C 180,E1 -26795.579,E2 -26795.579} C_VEL
LIN {X 0,Y 171.951,Z 443.407,A -85,B 0,C 180,E1 -26796.868,E2 -26796.868} C_VEL
LIN {X 0,Y 177.324,Z 428.321,A -85,B 0,C 180,E1 -26797.882,E2 -26797.882} C_VEL
LIN {X 0,Y 181.355,Z 413.384,A -85,B 0,C 180,E1 -26798.588,E2 -26798.588} C_VEL
LIN {X 0,Y 184.098,Z 398.526,A -85,B 0,C 180,E1 -26799.101,E2 -26799.101} C_VEL
LIN {X 0,Y 188.314,Z 358.219,A -85,B 0,C 180,E1 -26800.121,E2 -26800.121} C_VEL
LIN {X 0,Y 186.58,Z 352.49,A -85,B 0,C 180,E1 -26802.321,E2 -26802.321} C_VEL
LIN {X 0,Y 184.054,Z 346.782,A -85,B 0,C 180,E1 -26805.793,E2 -26805.793} C_VEL
LIN {X 0,Y 182.256,Z 343.115,A -85,B 0,C 180,E1 -26808.884,E2 -26808.884} C_VEL
LIN {X 0,Y 180.962,Z 340.176,A -85,B 0,C 180,E1 -26811.907,E2 -26811.907} C_VEL
LIN {X 0,Y 179.698,Z 336.66,A -85,B 0,C 180,E1 -26817.478,E2 -26817.478} C_VEL
LIN {X 0,Y 179.553,Z 336.173,A -85,B 0,C 180,E1 -26820,E2 -26820} C_VEL
LIN {X 0,Y 179.699,Z 336.623,A -85,B 0,C 180,E1 -26822.943,E2 -26822.943} C_VEL
LIN {X 0,Y 180.869,Z 340.088,A -85,B 0,C 180,E1 -26828.308,E2 -26828.308} C_VEL
LIN {X 0,Y 182.64,Z 343.832,A -85,B 0,C 180,E1 -26832.279,E2 -26832.279} C_VEL
LIN {X 0,Y 184.96,Z 348.821,A -85,B 0,C 180,E1 -26835.991,E2 -26835.991} C_VEL
LIN {X 0,Y 187.778,Z 355.306,A -85,B 0,C 180,E1 -26839.543,E2 -26839.543} C_VEL
LIN {X 0,Y 188.444,Z 356.904,A -85,B 0,C 180,E1 -26840.287,E2 -26840.287} C_VEL
LIN {X 0,Y 184.339,Z 395.516,A -85,B 0,C 180,E1 -26841.244,E2 -26841.244} C_VEL
LIN {X 0,Y 181.46,Z 410.943,A -85,B 0,C 180,E1 -26841.83,E2 -26841.83} C_VEL
LIN {X 0,Y 177.501,Z 425.628,A -85,B 0,C 180,E1 -26842.629,E2 -26842.629} C_VEL
LIN {X 0,Y 172.652,Z 439.413,A -85,B 0,C 180,E1 -26843.671,E2 -26843.671} C_VEL
LIN {X 0,Y 166.789,Z 452.997,A -85,B 0,C 180,E1 -26845.079,E2 -26845.079} C_VEL
LIN {X 0,Y 159.649,Z 466.672,A -85,B 0,C 180,E1 -26846.948,E2 -26846.948} C_VEL
LIN {X 0,Y 151.806,Z 479.073,A -85,B 0,C 180,E1 -26849.095,E2 -26849.095} C_VEL
LIN {X 0,Y 144.254,Z 489.453,A -85,B 0,C 180,E1 -26851.507,E2 -26851.507} C_VEL
LIN {X 0,Y 136.286,Z 499.082,A -85,B 0,C 180,E1 -26854.405,E2 -26854.405} C_VEL
LIN {X 0,Y 127.709,Z 508.508,A -85,B 0,C 180,E1 -26858.355,E2 -26858.355} C_VEL
LIN {X 0,Y 119.519,Z 516.361,A -85,B 0,C 180,E1 -26862.692,E2 -26862.692} C_VEL
LIN {X 0,Y 111.144,Z 523.684,A -85,B 0,C 180,E1 -26868.399,E2 -26868.399} C_VEL
LIN {X 0,Y 104.003,Z 529.485,A -85,B 0,C 180,E1 -26874.944,E2 -26874.944} C_VEL
LIN {X 0,Y 99.637,Z 532.914,A -85,B 0,C 180,E1 -26880.413,E2 -26880.413} C_VEL
LIN {X 0,Y 95.11,Z 536.38,A -85,B 0,C 180,E1 -26888.318,E2 -26888.318} C_VEL
LIN {X 0,Y 92.311,Z 538.659,A -85,B 0,C 180,E1 -26896.797,E2 -26896.797} C_VEL
LIN {X 0,Y 91.106,Z 539.813,A -85,B 0,C 180,E1 -26905.576,E2 -26905.576} C_VEL
LIN {X 0,Y 91.056,Z 539.964,A -85,B 0,C 180,E1 -26910,E2 -26910} C_VEL
LIN {X 0,Y 91.541,Z 539.404,A -85,B 0,C 180,E1 -26918.832,E2 -26918.832} C_VEL
LIN {X 0,Y 93.475,Z 537.734,A -85,B 0,C 180,E1 -26927.502,E2 -26927.502} C_VEL
LIN {X 0,Y 97.067,Z 534.908,A -85,B 0,C 180,E1 -26935.748,E2 -26935.748} C_VEL
LIN {X 0,Y 102.429,Z 530.851,A -85,B 0,C 180,E1 -26943.291,E2 -26943.291} C_VEL
LIN {X 0,Y 109.221,Z 525.467,A -85,B 0,C 180,E1 -26950.049,E2 -26950.049} C_VEL
LIN {X 0,Y 117.258,Z 518.599,A -85,B 0,C 180,E1 -26955.99,E2 -26955.99} C_VEL
LIN {X 0,Y 125.183,Z 511.215,A -85,B 0,C 180,E1 -26960.528,E2 -26960.528} C_VEL
LIN {X 0,Y 132.878,Z 503.152,A -85,B 0,C 180,E1 -26964.243,E2 -26964.243} C_VEL
LIN {X 0,Y 141.464,Z 493.219,A -85,B 0,C 180,E1 -26967.624,E2 -26967.624} C_VEL
LIN {X 0,Y 148.262,Z 484.433,A -85,B 0,C 180,E1 -26969.892,E2 -26969.892} C_VEL
LIN {X 0,Y 155.953,Z 473.109,A -85,B 0,C 180,E1 -26972.175,E2 -26972.175} C_VEL
LIN {X 0,Y 163.125,Z 460.801,A -85,B 0,C 180,E1 -26974.072,E2 -26974.072} C_VEL
LIN {X 0,Y 169.657,Z 447.336,A -85,B 0,C 180,E1 -26975.689,E2 -26975.689} C_VEL
LIN {X 0,Y 175.196,Z 433.37,A -85,B 0,C 180,E1 -26976.943,E2 -26976.943} C_VEL
LIN {X 0,Y 179.664,Z 419.01,A -85,B 0,C 180,E1 -26977.906,E2 -26977.906} C_VEL
LIN {X 0,Y 183.186,Z 403.876,A -85,B 0,C 180,E1 -26978.596,E2 -26978.596} C_VEL
LIN {X 0,Y 185.517,Z 388.296,A -85,B 0,C 180,E1 -26979.068,E2 -26979.068} C_VEL
LIN {X 0,Y 188.672,Z 356.981,A -85,B 0,C 180,E1 -26979.861,E2 -26979.861} C_VEL
LIN {X 0,Y 185.835,Z 350.455,A -85,B 0,C 180,E1 -26983.275,E2 -26983.275} C_VEL
LIN {X 0,Y 183.711,Z 345.82,A -85,B 0,C 180,E1 -26986.42,E2 -26986.42} C_VEL
LIN {X 0,Y 182.358,Z 343.042,A -85,B 0,C 180,E1 -26988.889,E2 -26988.889} C_VEL
LIN {X 0,Y 181.144,Z 340.253,A -85,B 0,C 180,E1 -26991.845,E2 -26991.845} C_VEL
LIN {X 0,Y 179.924,Z 336.411,A -85,B 0,C 180,E1 -26998.321,E2 -26998.321} C_VEL
LIN {X 0,Y 179.954,Z 336.423,A -85,B 0,C 180,E1 -27001.678,E2 -27001.678} C_VEL
LIN {X 0,Y 180.89,Z 339.906,A -85,B 0,C 180,E1 -27007.101,E2 -27007.101} C_VEL
LIN {X 0,Y 181.451,Z 340.897,A -85,B 0,C 180,E1 -27008.632,E2 -27008.632} C_VEL
LIN {X 0,Y 183.186,Z 344.697,A -85,B 0,C 180,E1 -27012.322,E2 -27012.322} C_VEL
LIN {X 0,Y 184.999,Z 348.576,A -85,B 0,C 180,E1 -27015.21,E2 -27015.21} C_VEL
LIN {X 0,Y 187.038,Z 353.298,A -85,B 0,C 180,E1 -27017.917,E2 -27017.917} C_VEL
LIN {X 0,Y 188.567,Z 358.445,A -85,B 0,C 180,E1 -27019.858,E2 -27019.858} C_VEL
LIN {X 0,Y 184.29,Z 399.07,A -85,B 0,C 180,E1 -27020.881,E2 -27020.881} C_VEL
LIN {X 0,Y 181.189,Z 415.128,A -85,B 0,C 180,E1 -27021.425,E2 -27021.425} C_VEL
LIN {X 0,Y 176.999,Z 430.339,A -85,B 0,C 180,E1 -27022.236,E2 -27022.236} C_VEL
LIN {X 0,Y 171.996,Z 444.052,A -85,B 0,C 180,E1 -27023.167,E2 -27023.167} C_VEL
LIN {X 0,Y 165.96,Z 457.492,A -85,B 0,C 180,E1 -27024.432,E2 -27024.432} C_VEL
LIN {X 0,Y 159.064,Z 470.398,A -85,B 0,C 180,E1 -27026.095,E2 -27026.095} C_VEL
LIN {X 0,Y 151.423,Z 482.519,A -85,B 0,C 180,E1 -27028.136,E2 -27028.136} C_VEL
LIN {X 0,Y 142.971,Z 493.992,A -85,B 0,C 180,E1 -27030.658,E2 -27030.658} C_VEL
LIN {X 0,Y 134.962,Z 503.657,A -85,B 0,C 180,E1 -27033.575,E2 -27033.575} C_VEL
LIN {X 0,Y 126.077,Z 513.156,A -85,B 0,C 180,E1 -27037.408,E2 -27037.408} C_VEL
LIN {X 0,Y 117.944,Z 521.08,A -85,B 0,C 180,E1 -27041.856,E2 -27041.856} C_VEL
LIN {X 0,Y 109.568,Z 528.483,A -85,B 0,C 180,E1 -27047.664,E2 -27047.664} C_VEL
LIN {X 0,Y 102.498,Z 534.365,A -85,B 0,C 180,E1 -27054.352,E2 -27054.352} C_VEL
LIN {X 0,Y 98.206,Z 537.872,A -85,B 0,C 180,E1 -27059.938,E2 -27059.938} C_VEL
LIN {X 0,Y 93.929,Z 541.419,A -85,B 0,C 180,E1 -27068.031,E2 -27068.031} C_VEL
LIN {X 0,Y 91.501,Z 543.763,A -85,B 0,C 180,E1 -27076.678,E2 -27076.678} C_VEL
LIN {X 0,Y 90.807,Z 544.952,A -85,B 0,C 180,E1 -27085.561,E2 -27085.561} C_VEL
LIN {X 0,Y 90.969,Z 545.114,A -85,B 0,C 180,E1 -27090,E2 -27090} C_VEL
LIN {X 0,Y 90.95,Z 544.48,A -85,B 0,C 180,E1 -27098.89,E2 -27098.89} C_VEL
LIN {X 0,Y 92.642,Z 542.465,A -85,B 0,C 180,E1 -27108.431,E2 -27108.431} C_VEL
LIN {X 0,Y 95.801,Z 539.728,A -85,B 0,C 180,E1 -27116.114,E2 -27116.114} C_VEL
LIN {X 0,Y 100.912,Z 535.529,A -85,B 0,C 180,E1 -27123.859,E2 -27123.859} C_VEL
LIN {X 0,Y 101.943,Z 534.69,A -85,B 0,C 180,E1 -27125.066,E2 -27125.066} C_VEL
LIN {X 0,Y 103.937,Z 532.683,A -85,B 0,C 180,E1 -27127.948,E2 -27127.948} C_VEL
LIN {X 0,Y 106.137,Z 529.112,A -85,B 0,C 180,E1 -27132.844,E2 -27132.844} C_VEL
LIN {X 0,Y 108.849,Z 525.054,A -85,B 0,C 180,E1 -27137.451,E2 -27137.451} C_VEL
LIN {X 0,Y 111.529,Z 522.266,A -85,B 0,C 180,E1 -27139.78,E2 -27139.78} C_VEL
LIN {X 0,Y 120.565,Z 513.993,A -85,B 0,C 180,E1 -27144.693,E2 -27144.693} C_VEL
LIN {X 0,Y 129.757,Z 504.709,A -85,B 0,C 180,E1 -27148.544,E2 -27148.544} C_VEL
LIN {X 0,Y 138.043,Z 495.28,A -85,B 0,C 180,E1 -27151.427,E2 -27151.427} C_VEL
LIN {X 0,Y 147.463,Z 483.05,A -85,B 0,C 180,E1 -27154.099,E2 -27154.099} C_VEL
LIN {X 0,Y 155.575,Z 470.575,A -85,B 0,C 180,E1 -27156.172,E2 -27156.172} C_VEL
LIN {X 0,Y 162.37,Z 458.314,A -85,B 0,C 180,E1 -27157.694,E2 -27157.694} C_VEL
LIN {X 0,Y 168.524,Z 445.051,A -85,B 0,C 180,E1 -27158.922,E2 -27158.922} C_VEL
LIN {X 0,Y 173.997,Z 430.532,A -85,B 0,C 180,E1 -27159.898,E2 -27159.898} C_VEL
LIN {X 0,Y 178.323,Z 415.465,A -85,B 0,C 180,E1 -27160.63,E2 -27160.63} C_VEL
LIN {X 0,Y 181.418,Z 400.017,A -85,B 0,C 180,E1 -27161.142,E2 -27161.142} C_VEL
LIN {X 0,Y 185.4,Z 364.29,A -85,B 0,C 180,E1 -27161.996,E2 -27161.996} C_VEL
LIN {X 0,Y 185.636,Z 361.498,A -85,B 0,C 180,E1 -27162.114,E2 -27162.114} C_VEL
LIN {X 0,Y 184.458,Z 357.728,A -85,B 0,C 180,E1 -27163.769,E2 -27163.769} C_VEL
LIN {X 0,Y 182.237,Z 352.531,A -85,B 0,C 180,E1 -27167.188,E2 -27167.188} C_VEL
LIN {X 0,Y 180.9,Z 349.537,A -85,B 0,C 180,E1 -27169.79,E2 -27169.79} C_VEL
LIN {X 0,Y 179.881,Z 347.038,A -85,B 0,C 180,E1 -27172.423,E2 -27172.423} C_VEL
LIN {X 0,Y 178.758,Z 343.413,A -85,B 0,C 180,E1 -27178.347,E2 -27178.347} C_VEL
LIN {X 0,Y 178.697,Z 343.31,A -85,B 0,C 180,E1 -27181.127,E2 -27181.127} C_VEL
LIN {X 0,Y 178.802,Z 343.773,A -85,B 0,C 180,E1 -27182.816,E2 -27182.816} C_VEL
LIN {X 0,Y 180.136,Z 347.701,A -85,B 0,C 180,E1 -27188.766,E2 -27188.766} C_VEL
LIN {X 0,Y 181.774,Z 351.52,A -85,B 0,C 180,E1 -27192.424,E2 -27192.424} C_VEL
LIN {X 0,Y 183.752,Z 356.044,A -85,B 0,C 180,E1 -27195.672,E2 -27195.672} C_VEL
LIN {X 0,Y 185.71,Z 360.853,A -85,B 0,C 180,E1 -27198.321,E2 -27198.321} C_VEL
LIN {X 0,Y 181.785,Z 396.347,A -85,B 0,C 180,E1 -27199.179,E2 -27199.179} C_VEL
LIN {X 0,Y 178.755,Z 411.919,A -85,B 0,C 180,E1 -27199.76,E2 -27199.76} C_VEL
LIN {X 0,Y 174.516,Z 426.984,A -85,B 0,C 180,E1 -27200.562,E2 -27200.562} C_VEL
LIN {X 0,Y 169.169,Z 441.474,A -85,B 0,C 180,E1 -27201.638,E2 -27201.638} C_VEL
LIN {X 0,Y 163.011,Z 455.059,A -85,B 0,C 180,E1 -27203.056,E2 -27203.056} C_VEL
LIN {X 0,Y 155.818,Z 468.113,A -85,B 0,C 180,E1 -27204.811,E2 -27204.811} C_VEL
LIN {X 0,Y 147.772,Z 480.31,A -85,B 0,C 180,E1 -27206.91,E2 -27206.91} C_VEL
LIN {X 0,Y 139.256,Z 491.422,A -85,B 0,C 180,E1 -27209.477,E2 -27209.477} C_VEL
LIN {X 0,Y 130.199,Z 501.676,A -85,B 0,C 180,E1 -27212.67,E2 -27212.67} C_VEL
LIN {X 0,Y 122.136,Z 509.935,A -85,B 0,C 180,E1 -27216.334,E2 -27216.334} C_VEL
LIN {X 0,Y 113.639,Z 517.564,A -85,B 0,C 180,E1 -27220.748,E2 -27220.748} C_VEL
LIN {X 0,Y 105.922,Z 523.887,A -85,B 0,C 180,E1 -27225.84,E2 -27225.84} C_VEL
LIN {X 0,Y 98.248,Z 529.688,A -85,B 0,C 180,E1 -27232.554,E2 -27232.554} C_VEL
LIN {X 0,Y 93.497,Z 533.117,A -85,B 0,C 180,E1 -27238.253,E2 -27238.253} C_VEL
LIN {X 0,Y 88.518,Z 536.582,A -85,B 0,C 180,E1 -27246.611,E2 -27246.611} C_VEL
LIN {X 0,Y 85.405,Z 538.861,A -85,B 0,C 180,E1 -27255.708,E2 -27255.708} C_VEL
LIN {X 0,Y 84.05,Z 540.013,A -85,B 0,C 180,E1 -27265.204,E2 -27265.204} C_VEL
LIN {X 0,Y 83.956,Z 540.165,A -85,B 0,C 180,E1 -27270,E2 -27270} C_VEL
LIN {X 0,Y 84.513,Z 539.605,A -85,B 0,C 180,E1 -27279.573,E2 -27279.573} C_VEL
LIN {X 0,Y 86.703,Z 537.935,A -85,B 0,C 180,E1 -27288.919,E2 -27288.919} C_VEL
LIN {X 0,Y 90.693,Z 535.11,A -85,B 0,C 180,E1 -27297.706,E2 -27297.706} C_VEL
LIN {X 0,Y 96.539,Z 531.052,A -85,B 0,C 180,E1 -27305.618,E2 -27305.618} C_VEL
LIN {X 0,Y 103.86,Z 525.667,A -85,B 0,C 180,E1 -27312.583,E2 -27312.583} C_VEL
LIN {X 0,Y 112.41,Z 518.8,A -85,B 0,C 180,E1 -27318.611,E2 -27318.611} C_VEL
LIN {X 0,Y 120.79,Z 511.414,A -85,B 0,C 180,E1 -27323.131,E2 -27323.131} C_VEL
LIN {X 0,Y 129.398,Z 502.729,A -85,B 0,C 180,E1 -27327.103,E2 -27327.103} C_VEL
LIN {X 0,Y 137.792,Z 493.417,A -85,B 0,C 180,E1 -27330.118,E2 -27330.118} C_VEL
LIN {X 0,Y 146.234,Z 482.688,A -85,B 0,C 180,E1 -27332.759,E2 -27332.759} C_VEL
LIN {X 0,Y 154.233,Z 470.968,A -85,B 0,C 180,E1 -27334.908,E2 -27334.908} C_VEL
LIN {X 0,Y 160.891,Z 459.584,A -85,B 0,C 180,E1 -27336.534,E2 -27336.534} C_VEL
LIN {X 0,Y 166.861,Z 447.532,A -85,B 0,C 180,E1 -27337.909,E2 -27337.909} C_VEL
LIN {X 0,Y 172.545,Z 433.564,A -85,B 0,C 180,E1 -27339.108,E2 -27339.108} C_VEL
LIN {X 0,Y 177.121,Z 419.202,A -85,B 0,C 180,E1 -27340.031,E2 -27340.031} C_VEL
LIN {X 0,Y 180.848,Z 403.449,A -85,B 0,C 180,E1 -27340.713,E2 -27340.713} C_VEL
LIN {X 0,Y 183.272,Z 386.934,A -85,B 0,C 180,E1 -27341.183,E2 -27341.183} C_VEL
LIN {X 0,Y 185.945,Z 360.962,A -85,B 0,C 180,E1 -27341.826,E2 -27341.826} C_VEL
LIN {X 0,Y 183.552,Z 355.161,A -85,B 0,C 180,E1 -27345.143,E2 -27345.143} C_VEL
LIN {X 0,Y 181.546,Z 350.485,A -85,B 0,C 180,E1 -27348.698,E2 -27348.698} C_VEL
LIN {X 0,Y 180.05,Z 347.071,A -85,B 0,C 180,E1 -27352.43,E2 -27352.43} C_VEL
LIN {X 0,Y 179.056,Z 343.479,A -85,B 0,C 180,E1 -27358.313,E2 -27358.313} C_VEL
LIN {X 0,Y 179.054,Z 343.365,A -85,B 0,C 180,E1 -27361.124,E2 -27361.124} C_VEL
LIN {X 0,Y 180.358,Z 347.739,A -85,B 0,C 180,E1 -27368.12,E2 -27368.12} C_VEL
LIN {X 0,Y 181.971,Z 351.519,A -85,B 0,C 180,E1 -27371.804,E2 -27371.804} C_VEL
LIN {X 0,Y 183.986,Z 356.147,A -85,B 0,C 180,E1 -27375.154,E2 -27375.154} C_VEL
LIN {X 0,Y 185.282,Z 359.595,A -85,B 0,C 180,E1 -27377.003,E2 -27377.003} C_VEL
LIN {X 0,Y 185.911,Z 361.874,A -85,B 0,C 180,E1 -27377.9,E2 -27377.9} C_VEL
LIN {X 0,Y 181.882,Z 398.885,A -85,B 0,C 180,E1 -27378.793,E2 -27378.793} C_VEL
LIN {X 0,Y 178.718,Z 414.936,A -85,B 0,C 180,E1 -27379.306,E2 -27379.306} C_VEL
LIN {X 0,Y 174.437,Z 430.145,A -85,B 0,C 180,E1 -27380.078,E2 -27380.078} C_VEL
LIN {X 0,Y 169.319,Z 443.857,A -85,B 0,C 180,E1 -27380.95,E2 -27380.95} C_VEL
LIN {X 0,Y 163.149,Z 457.296,A -85,B 0,C 180,E1 -27382.159,E2 -27382.159} C_VEL
LIN {X 0,Y 155.604,Z 470.988,A -85,B 0,C 180,E1 -27383.853,E2 -27383.853} C_VEL
LIN {X 0,Y 147.461,Z 483.392,A -85,B 0,C 180,E1 -27385.9,E2 -27385.9} C_VEL
LIN {X 0,Y 138.054,Z 495.552,A -85,B 0,C 180,E1 -27388.582,E2 -27388.582} C_VEL
LIN {X 0,Y 128.437,Z 506.382,A -85,B 0,C 180,E1 -27391.991,E2 -27391.991} C_VEL
LIN {X 0,Y 119.302,Z 515.431,A -85,B 0,C 180,E1 -27395.934,E2 -27395.934} C_VEL
LIN {X 0,Y 111.015,Z 522.912,A -85,B 0,C 180,E1 -27400.565,E2 -27400.565} C_VEL
LIN {X 0,Y 102.345,Z 529.909,A -85,B 0,C 180,E1 -27406.632,E2 -27406.632} C_VEL
LIN {X 0,Y 95.076,Z 535.42,A -85,B 0,C 180,E1 -27413.748,E2 -27413.748} C_VEL
LIN {X 0,Y 89.457,Z 539.597,A -85,B 0,C 180,E1 -27421.877,E2 -27421.877} C_VEL
LIN {X 0,Y 85.648,Z 542.534,A -85,B 0,C 180,E1 -27430.839,E2 -27430.839} C_VEL
LIN {X 0,Y 83.9,Z 544.299,A -85,B 0,C 180,E1 -27440.356,E2 -27440.356} C_VEL
LIN {X 0,Y 83.875,Z 544.913,A -85,B 0,C 180,E1 -27450,E2 -27450} C_VEL
LIN {X 0,Y 83.728,Z 544.744,A -85,B 0,C 180,E1 -27454.815,E2 -27454.815} C_VEL
LIN {X 0,Y 84.552,Z 543.526,A -85,B 0,C 180,E1 -27464.439,E2 -27464.439} C_VEL
LIN {X 0,Y 87.29,Z 541.154,A -85,B 0,C 180,E1 -27473.738,E2 -27473.738} C_VEL
LIN {X 0,Y 91.986,Z 537.584,A -85,B 0,C 180,E1 -27482.331,E2 -27482.331} C_VEL
LIN {X 0,Y 98.501,Z 532.73,A -85,B 0,C 180,E1 -27489.951,E2 -27489.951} C_VEL
LIN {X 0,Y 106.503,Z 526.46,A -85,B 0,C 180,E1 -27496.54,E2 -27496.54} C_VEL
LIN {X 0,Y 111.529,Z 522.266,A -85,B 0,C 180,E1 -27499.78,E2 -27499.78} C_VEL
LIN {X 0,Y 114.327,Z 519.404,A -85,B 0,C 180,E1 -27501.974,E2 -27501.974} C_VEL
LIN {X 0,Y 121.028,Z 510.294,A -85,B 0,C 180,E1 -27508.716,E2 -27508.716} C_VEL
LIN {X 0,Y 123.966,Z 506.827,A -85,B 0,C 180,E1 -27510.472,E2 -27510.472} C_VEL
LIN {X 0,Y 125.115,Z 505.6,A -85,B 0,C 180,E1 -27510.94,E2 -27510.94} C_VEL
LIN {X 0,Y 134.768,Z 495.075,A -85,B 0,C 180,E1 -27514.099,E2 -27514.099} C_VEL
LIN {X 0,Y 144.487,Z 482.844,A -85,B 0,C 180,E1 -27516.647,E2 -27516.647} C_VEL
LIN {X 0,Y 152.83,Z 470.369,A -85,B 0,C 180,E1 -27518.621,E2 -27518.621} C_VEL
LIN {X 0,Y 159.8,Z 458.108,A -85,B 0,C 180,E1 -27520.06,E2 -27520.06} C_VEL
LIN {X 0,Y 166.096,Z 444.844,A -85,B 0,C 180,E1 -27521.214,E2 -27521.214} C_VEL
LIN {X 0,Y 171.685,Z 430.324,A -85,B 0,C 180,E1 -27522.124,E2 -27522.124} C_VEL
LIN {X 0,Y 176.098,Z 415.254,A -85,B 0,C 180,E1 -27522.807,E2 -27522.807} C_VEL
LIN {X 0,Y 179.166,Z 400.269,A -85,B 0,C 180,E1 -27523.279,E2 -27523.279} C_VEL
LIN {X 0,Y 182.532,Z 371.518,A -85,B 0,C 180,E1 -27523.94,E2 -27523.94} C_VEL
LIN {X 0,Y 183.201,Z 365.147,A -85,B 0,C 180,E1 -27524.097,E2 -27524.097} C_VEL
LIN {X 0,Y 181.364,Z 360.239,A -85,B 0,C 180,E1 -27527.055,E2 -27527.055} C_VEL
LIN {X 0,Y 179.75,Z 356.322,A -85,B 0,C 180,E1 -27530.329,E2 -27530.329} C_VEL
LIN {X 0,Y 178.792,Z 353.861,A -85,B 0,C 180,E1 -27533.015,E2 -27533.015} C_VEL
LIN {X 0,Y 177.891,Z 350.475,A -85,B 0,C 180,E1 -27538.339,E2 -27538.339} C_VEL
LIN {X 0,Y 177.861,Z 350.426,A -85,B 0,C 180,E1 -27541.698,E2 -27541.698} C_VEL
LIN {X 0,Y 179.029,Z 354.473,A -85,B 0,C 180,E1 -27548.181,E2 -27548.181} C_VEL
LIN {X 0,Y 180.428,Z 357.995,A -85,B 0,C 180,E1 -27551.616,E2 -27551.616} C_VEL
LIN {X 0,Y 182.184,Z 362.319,A -85,B 0,C 180,E1 -27554.772,E2 -27554.772} C_VEL
LIN {X 0,Y 183.165,Z 364.956,A -85,B 0,C 180,E1 -27556.281,E2 -27556.281} C_VEL
LIN {X 0,Y 179.551,Z 396.739,A -85,B 0,C 180,E1 -27557.048,E2 -27557.048} C_VEL
LIN {X 0,Y 176.484,Z 412.129,A -85,B 0,C 180,E1 -27557.594,E2 -27557.594} C_VEL
LIN {X 0,Y 172.156,Z 427.191,A -85,B 0,C 180,E1 -27558.355,E2 -27558.355} C_VEL
LIN {X 0,Y 166.689,Z 441.68,A -85,B 0,C 180,E1 -27559.376,E2 -27559.376} C_VEL
LIN {X 0,Y 160.675,Z 454.657,A -85,B 0,C 180,E1 -27560.641,E2 -27560.641} C_VEL
LIN {X 0,Y 152.975,Z 468.317,A -85,B 0,C 180,E1 -27562.397,E2 -27562.397} C_VEL
LIN {X 0,Y 144.684,Z 480.515,A -85,B 0,C 180,E1 -27564.39,E2 -27564.39} C_VEL
LIN {X 0,Y 135.904,Z 491.626,A -85,B 0,C 180,E1 -27566.871,E2 -27566.871} C_VEL
LIN {X 0,Y 126.084,Z 502.303,A -85,B 0,C 180,E1 -27570.111,E2 -27570.111} C_VEL
LIN {X 0,Y 118.056,Z 510.138,A -85,B 0,C 180,E1 -27573.549,E2 -27573.549} C_VEL
LIN {X 0,Y 109.116,Z 517.767,A -85,B 0,C 180,E1 -27577.909,E2 -27577.909} C_VEL
LIN {X 0,Y 100.918,Z 524.09,A -85,B 0,C 180,E1 -27583.012,E2 -27583.012} C_VEL
LIN {X 0,Y 92.688,Z 529.891,A -85,B 0,C 180,E1 -27589.872,E2 -27589.872} C_VEL
LIN {X 0,Y 87.513,Z 533.32,A -85,B 0,C 180,E1 -27595.796,E2 -27595.796} C_VEL
LIN {X 0,Y 82.024,Z 536.784,A -85,B 0,C 180,E1 -27604.634,E2 -27604.634} C_VEL
LIN {X 0,Y 78.521,Z 539.063,A -85,B 0,C 180,E1 -27614.425,E2 -27614.425} C_VEL
LIN {X 0,Y 76.987,Z 540.214,A -85,B 0,C 180,E1 -27624.762,E2 -27624.762} C_VEL
LIN {X 0,Y 76.883,Z 540.365,A -85,B 0,C 180,E1 -27630,E2 -27630} C_VEL
LIN {X 0,Y 77.511,Z 539.806,A -85,B 0,C 180,E1 -27640.448,E2 -27640.448} C_VEL
LIN {X 0,Y 80.002,Z 538.136,A -85,B 0,C 180,E1 -27650.572,E2 -27650.572} C_VEL
LIN {X 0,Y 84.447,Z 535.311,A -85,B 0,C 180,E1 -27659.956,E2 -27659.956} C_VEL
LIN {X 0,Y 90.836,Z 531.253,A -85,B 0,C 180,E1 -27668.239,E2 -27668.239} C_VEL
LIN {X 0,Y 98.717,Z 525.868,A -85,B 0,C 180,E1 -27675.391,E2 -27675.391} C_VEL
LIN {X 0,Y 107.827,Z 519,A -85,B 0,C 180,E1 -27681.455,E2 -27681.455} C_VEL
LIN {X 0,Y 116.66,Z 511.613,A -85,B 0,C 180,E1 -27685.927,E2 -27685.927} C_VEL
LIN {X 0,Y 126.111,Z 502.509,A -85,B 0,C 180,E1 -27689.981,E2 -27689.981} C_VEL
LIN {X 0,Y 135.85,Z 491.995,A -85,B 0,C 180,E1 -27693.174,E2 -27693.174} C_VEL
LIN {X 0,Y 145.364,Z 479.946,A -85,B 0,C 180,E1 -27695.859,E2 -27695.859} C_VEL
LIN {X 0,Y 153.67,Z 467.635,A -85,B 0,C 180,E1 -27697.834,E2 -27697.834} C_VEL
LIN {X 0,Y 161.318,Z 453.858,A -85,B 0,C 180,E1 -27699.602,E2 -27699.602} C_VEL
LIN {X 0,Y 167.409,Z 440.685,A -85,B 0,C 180,E1 -27700.83,E2 -27700.83} C_VEL
LIN {X 0,Y 172.893,Z 425.876,A -85,B 0,C 180,E1 -27701.834,E2 -27701.834} C_VEL
LIN {X 0,Y 177.191,Z 410.233,A -85,B 0,C 180,E1 -27702.634,E2 -27702.634} C_VEL
LIN {X 0,Y 180.089,Z 395.165,A -85,B 0,C 180,E1 -27703.113,E2 -27703.113} C_VEL
LIN {X 0,Y 183.425,Z 365.08,A -85,B 0,C 180,E1 -27703.849,E2 -27703.849} C_VEL
LIN {X 0,Y 181.304,Z 359.606,A -85,B 0,C 180,E1 -27707.334,E2 -27707.334} C_VEL
LIN {X 0,Y 179.953,Z 356.458,A -85,B 0,C 180,E1 -27710.162,E2 -27710.162} C_VEL
LIN {X 0,Y 178.996,Z 353.937,A -85,B 0,C 180,E1 -27712.952,E2 -27712.952} C_VEL
LIN {X 0,Y 178.162,Z 350.453,A -85,B 0,C 180,E1 -27718.87,E2 -27718.87} C_VEL
LIN {X 0,Y 178.174,Z 350.531,A -85,B 0,C 180,E1 -27721.13,E2 -27721.13} C_VEL
LIN {X 0,Y 179.321,Z 354.697,A -85,B 0,C 180,E1 -27727.73,E2 -27727.73} C_VEL
LIN {X 0,Y 180.674,Z 358.124,A -85,B 0,C 180,E1 -27731.085,E2 -27731.085} C_VEL
LIN {X 0,Y 182.42,Z 362.443,A -85,B 0,C 180,E1 -27734.253,E2 -27734.253} C_VEL
LIN {X 0,Y 183.452,Z 365.413,A -85,B 0,C 180,E1 -27735.874,E2 -27735.874} C_VEL
LIN {X 0,Y 179.643,Z 399.171,A -85,B 0,C 180,E1 -27736.663,E2 -27736.663} C_VEL
LIN {X 0,Y 176.506,Z 414.746,A -85,B 0,C 180,E1 -27737.139,E2 -27737.139} C_VEL
LIN {X 0,Y 172.126,Z 429.951,A -85,B 0,C 180,E1 -27737.854,E2 -27737.854} C_VEL
LIN {X 0,Y 166.906,Z 443.661,A -85,B 0,C 180,E1 -27738.667,E2 -27738.667} C_VEL
LIN {X 0,Y 160.598,Z 457.099,A -85,B 0,C 180,E1 -27739.805,E2 -27739.805} C_VEL
LIN {X 0,Y 152.852,Z 470.789,A -85,B 0,C 180,E1 -27741.4,E2 -27741.4} C_VEL
LIN {X 0,Y 144.488,Z 483.194,A -85,B 0,C 180,E1 -27743.354,E2 -27743.354} C_VEL
LIN {X 0,Y 134.777,Z 495.352,A -85,B 0,C 180,E1 -27745.91,E2 -27745.91} C_VEL
LIN {X 0,Y 124.784,Z 506.181,A -85,B 0,C 180,E1 -27749.196,E2 -27749.196} C_VEL
LIN {X 0,Y 116.591,Z 513.994,A -85,B 0,C 180,E1 -27752.447,E2 -27752.447} C_VEL
LIN {X 0,Y 107.661,Z 521.693,A -85,B 0,C 180,E1 -27756.903,E2 -27756.903} C_VEL
LIN {X 0,Y 99.436,Z 528.08,A -85,B 0,C 180,E1 -27762.089,E2 -27762.089} C_VEL
LIN {X 0,Y 91.225,Z 533.961,A -85,B 0,C 180,E1 -27769.093,E2 -27769.093} C_VEL
LIN {X 0,Y 86.065,Z 537.466,A -85,B 0,C 180,E1 -27775.138,E2 -27775.138} C_VEL
LIN {X 0,Y 80.808,Z 541.014,A -85,B 0,C 180,E1 -27784.224,E2 -27784.224} C_VEL
LIN {X 0,Y 77.637,Z 543.359,A -85,B 0,C 180,E1 -27794.243,E2 -27794.243} C_VEL
LIN {X 0,Y 76.621,Z 544.55,A -85,B 0,C 180,E1 -27804.737,E2 -27804.737} C_VEL
LIN {X 0,Y 76.771,Z 544.712,A -85,B 0,C 180,E1 -27810,E2 -27810} C_VEL
LIN {X 0,Y 76.878,Z 544.076,A -85,B 0,C 180,E1 -27820.535,E2 -27820.535} C_VEL
LIN {X 0,Y 78.896,Z 542.282,A -85,B 0,C 180,E1 -27830.874,E2 -27830.874} C_VEL
LIN {X 0,Y 83.149,Z 539.32,A -85,B 0,C 180,E1 -27840.473,E2 -27840.473} C_VEL
LIN {X 0,Y 89.359,Z 535.121,A -85,B 0,C 180,E1 -27848.99,E2 -27848.99} C_VEL
LIN {X 0,Y 97.249,Z 529.577,A -85,B 0,C 180,E1 -27856.275,E2 -27856.275} C_VEL
LIN {X 0,Y 106.471,Z 522.54,A -85,B 0,C 180,E1 -27862.381,E2 -27862.381} C_VEL
LIN {X 0,Y 115.354,Z 514.93,A -85,B 0,C 180,E1 -27867.015,E2 -27867.015} C_VEL
LIN {X 0,Y 125.115,Z 505.6,A -85,B 0,C 180,E1 -27870.94,E2 -27870.94} C_VEL
LIN {X 0,Y 128.322,Z 501.92,A -85,B 0,C 180,E1 -27872.416,E2 -27872.416} C_VEL
LIN {X 0,Y 136.012,Z 490.546,A -85,B 0,C 180,E1 -27877.353,E2 -27877.353} C_VEL
LIN {X 0,Y 138.981,Z 486.347,A -85,B 0,C 180,E1 -27878.583,E2 -27878.583} C_VEL
LIN {X 0,Y 140.097,Z 484.879,A -85,B 0,C 180,E1 -27878.887,E2 -27878.887} C_VEL
LIN {X 0,Y 148.817,Z 472.579,A -85,B 0,C 180,E1 -27880.821,E2 -27880.821} C_VEL
LIN {X 0,Y 155.919,Z 460.763,A -85,B 0,C 180,E1 -27882.209,E2 -27882.209} C_VEL
LIN {X 0,Y 163.142,Z 446.407,A -85,B 0,C 180,E1 -27883.433,E2 -27883.433} C_VEL
LIN {X 0,Y 168.831,Z 432.375,A -85,B 0,C 180,E1 -27884.283,E2 -27884.283} C_VEL
LIN {X 0,Y 173.52,Z 417.333,A -85,B 0,C 180,E1 -27884.953,E2 -27884.953} C_VEL
LIN {X 0,Y 176.908,Z 401.986,A -85,B 0,C 180,E1 -27885.429,E2 -27885.429} C_VEL
LIN {X 0,Y 179.636,Z 381.023,A -85,B 0,C 180,E1 -27885.889,E2 -27885.889} C_VEL
LIN {X 0,Y 180.894,Z 369.309,A -85,B 0,C 180,E1 -27886.172,E2 -27886.172} C_VEL
LIN {X 0,Y 179.414,Z 365.271,A -85,B 0,C 180,E1 -27888.991,E2 -27888.991} C_VEL
LIN {X 0,Y 178.422,Z 362.704,A -85,B 0,C 180,E1 -27891.363,E2 -27891.363} C_VEL
LIN {X 0,Y 177.767,Z 360.734,A -85,B 0,C 180,E1 -27893.474,E2 -27893.474} C_VEL
LIN {X 0,Y 176.991,Z 357.413,A -85,B 0,C 180,E1 -27898.887,E2 -27898.887} C_VEL
LIN {X 0,Y 176.993,Z 357.496,A -85,B 0,C 180,E1 -27901.707,E2 -27901.707} C_VEL
LIN {X 0,Y 177.963,Z 361.306,A -85,B 0,C 180,E1 -27907.66,E2 -27907.66} C_VEL
LIN {X 0,Y 179.342,Z 365.098,A -85,B 0,C 180,E1 -27911.3,E2 -27911.3} C_VEL
LIN {X 0,Y 180.878,Z 369.33,A -85,B 0,C 180,E1 -27914.254,E2 -27914.254} C_VEL
LIN {X 0,Y 177.579,Z 397.089,A -85,B 0,C 180,E1 -27914.866,E2 -27914.866} C_VEL
LIN {X 0,Y 174.472,Z 412.339,A -85,B 0,C 180,E1 -27915.374,E2 -27915.374} C_VEL
LIN {X 0,Y 170.06,Z 427.399,A -85,B 0,C 180,E1 -27916.091,E2 -27916.091} C_VEL
LIN {X 0,Y 164.472,Z 441.887,A -85,B 0,C 180,E1 -27917.044,E2 -27917.044} C_VEL
LIN {X 0,Y 157.976,Z 455.481,A -85,B 0,C 180,E1 -27918.303,E2 -27918.303} C_VEL
LIN {X 0,Y 150.41,Z 468.522,A -85,B 0,C 180,E1 -27919.893,E2 -27919.893} C_VEL
LIN {X 0,Y 141.893,Z 480.719,A -85,B 0,C 180,E1 -27921.772,E2 -27921.772} C_VEL
LIN {X 0,Y 132.84,Z 491.83,A -85,B 0,C 180,E1 -27924.132,E2 -27924.132} C_VEL
LIN {X 0,Y 123.791,Z 501.387,A -85,B 0,C 180,E1 -27926.864,E2 -27926.864} C_VEL
LIN {X 0,Y 114.275,Z 510.342,A -85,B 0,C 180,E1 -27930.572,E2 -27930.572} C_VEL
LIN {X 0,Y 104.892,Z 517.97,A -85,B 0,C 180,E1 -27934.839,E2 -27934.839} C_VEL
LIN {X 0,Y 96.201,Z 524.293,A -85,B 0,C 180,E1 -27939.909,E2 -27939.909} C_VEL
LIN {X 0,Y 88.11,Z 529.63,A -85,B 0,C 180,E1 -27946.126,E2 -27946.126} C_VEL
LIN {X 0,Y 81.715,Z 533.522,A -85,B 0,C 180,E1 -27952.984,E2 -27952.984} C_VEL
LIN {X 0,Y 75.628,Z 536.987,A -85,B 0,C 180,E1 -27962.314,E2 -27962.314} C_VEL
LIN {X 0,Y 71.696,Z 539.264,A -85,B 0,C 180,E1 -27972.898,E2 -27972.898} C_VEL
LIN {X 0,Y 69.918,Z 540.415,A -85,B 0,C 180,E1 -27984.231,E2 -27984.231} C_VEL
LIN {X 0,Y 69.783,Z 540.566,A -85,B 0,C 180,E1 -27990,E2 -27990} C_VEL
LIN {X 0,Y 70.543,Z 540.007,A -85,B 0,C 180,E1 -28001.493,E2 -28001.493} C_VEL
LIN {X 0,Y 73.369,Z 538.337,A -85,B 0,C 180,E1 -28012.529,E2 -28012.529} C_VEL
LIN {X 0,Y 78.356,Z 535.511,A -85,B 0,C 180,E1 -28022.557,E2 -28022.557} C_VEL
LIN {X 0,Y 85.35,Z 531.454,A -85,B 0,C 180,E1 -28031.203,E2 -28031.203} C_VEL
LIN {X 0,Y 93.83,Z 526.069,A -85,B 0,C 180,E1 -28038.503,E2 -28038.503} C_VEL
LIN {X 0,Y 103.541,Z 519.2,A -85,B 0,C 180,E1 -28044.538,E2 -28044.538} C_VEL
LIN {X 0,Y 112.828,Z 511.813,A -85,B 0,C 180,E1 -28048.922,E2 -28048.922} C_VEL
LIN {X 0,Y 122.404,Z 502.986,A -85,B 0,C 180,E1 -28052.763,E2 -28052.763} C_VEL
LIN {X 0,Y 131.289,Z 493.814,A -85,B 0,C 180,E1 -28055.505,E2 -28055.505} C_VEL
LIN {X 0,Y 140.297,Z 483.084,A -85,B 0,C 180,E1 -28057.928,E2 -28057.928} C_VEL
LIN {X 0,Y 148.779,Z 471.361,A -85,B 0,C 180,E1 -28059.856,E2 -28059.856} C_VEL
LIN {X 0,Y 156.446,Z 458.764,A -85,B 0,C 180,E1 -28061.47,E2 -28061.47} C_VEL
LIN {X 0,Y 162.835,Z 446.177,A -85,B 0,C 180,E1 -28062.727,E2 -28062.727} C_VEL
LIN {X 0,Y 168.799,Z 431.743,A -85,B 0,C 180,E1 -28063.779,E2 -28063.779} C_VEL
LIN {X 0,Y 173.413,Z 417.432,A -85,B 0,C 180,E1 -28064.531,E2 -28064.531} C_VEL
LIN {X 0,Y 176.787,Z 403.232,A -85,B 0,C 180,E1 -28065.077,E2 -28065.077} C_VEL
LIN {X 0,Y 179.11,Z 388.139,A -85,B 0,C 180,E1 -28065.458,E2 -28065.458} C_VEL
LIN {X 0,Y 181.121,Z 369.433,A -85,B 0,C 180,E1 -28065.911,E2 -28065.911} C_VEL
LIN {X 0,Y 179.597,Z 365.268,A -85,B 0,C 180,E1 -28068.859,E2 -28068.859} C_VEL
LIN {X 0,Y 178.534,Z 362.5,A -85,B 0,C 180,E1 -28071.511,E2 -28071.511} C_VEL
LIN {X 0,Y 177.924,Z 360.685,A -85,B 0,C 180,E1 -28073.617,E2 -28073.617} C_VEL
LIN {X 0,Y 177.292,Z 357.544,A -85,B 0,C 180,E1 -28078.864,E2 -28078.864} C_VEL
LIN {X 0,Y 177.294,Z 357.443,A -85,B 0,C 180,E1 -28080.568,E2 -28080.568} C_VEL
LIN {X 0,Y 178.256,Z 361.564,A -85,B 0,C 180,E1 -28087.219,E2 -28087.219} C_VEL
LIN {X 0,Y 179.397,Z 364.701,A -85,B 0,C 180,E1 -28090.332,E2 -28090.332} C_VEL
LIN {X 0,Y 180.934,Z 368.889,A -85,B 0,C 180,E1 -28093.405,E2 -28093.405} C_VEL
LIN {X 0,Y 181.16,Z 369.553,A -85,B 0,C 180,E1 -28093.806,E2 -28093.806} C_VEL
LIN {X 0,Y 177.612,Z 399.701,A -85,B 0,C 180,E1 -28094.491,E2 -28094.491} C_VEL
LIN {X 0,Y 174.336,Z 415.317,A -85,B 0,C 180,E1 -28094.933,E2 -28094.933} C_VEL
LIN {X 0,Y 170.08,Z 429.757,A -85,B 0,C 180,E1 -28095.573,E2 -28095.573} C_VEL
LIN {X 0,Y 164.769,Z 443.466,A -85,B 0,C 180,E1 -28096.325,E2 -28096.325} C_VEL
LIN {X 0,Y 158.332,Z 456.903,A -85,B 0,C 180,E1 -28097.386,E2 -28097.386} C_VEL
LIN {X 0,Y 150.392,Z 470.591,A -85,B 0,C 180,E1 -28098.865,E2 -28098.865} C_VEL
LIN {X 0,Y 141.805,Z 482.995,A -85,B 0,C 180,E1 -28100.701,E2 -28100.701} C_VEL
LIN {X 0,Y 131.817,Z 495.153,A -85,B 0,C 180,E1 -28103.12,E2 -28103.12} C_VEL
LIN {X 0,Y 121.45,Z 505.981,A -85,B 0,C 180,E1 -28106.244,E2 -28106.244} C_VEL
LIN {X 0,Y 111.583,Z 514.958,A -85,B 0,C 180,E1 -28109.923,E2 -28109.923} C_VEL
LIN {X 0,Y 102.237,Z 522.508,A -85,B 0,C 180,E1 -28114.423,E2 -28114.423} C_VEL
LIN {X 0,Y 92.432,Z 529.505,A -85,B 0,C 180,E1 -28120.507,E2 -28120.507} C_VEL
LIN {X 0,Y 83.955,Z 535.017,A -85,B 0,C 180,E1 -28127.958,E2 -28127.958} C_VEL
LIN {X 0,Y 77.1,Z 539.193,A -85,B 0,C 180,E1 -28136.845,E2 -28136.845} C_VEL
LIN {X 0,Y 72.263,Z 542.13,A -85,B 0,C 180,E1 -28147.107,E2 -28147.107} C_VEL
LIN {X 0,Y 69.861,Z 543.895,A -85,B 0,C 180,E1 -28158.393,E2 -28158.393} C_VEL
LIN {X 0,Y 69.666,Z 544.511,A -85,B 0,C 180,E1 -28170,E2 -28170} C_VEL
LIN {X 0,Y 69.858,Z 543.873,A -85,B 0,C 180,E1 -28181.607,E2 -28181.607} C_VEL
LIN {X 0,Y 72.244,Z 542.078,A -85,B 0,C 180,E1 -28192.9,E2 -28192.9} C_VEL
LIN {X 0,Y 77.052,Z 539.116,A -85,B 0,C 180,E1 -28203.179,E2 -28203.179} C_VEL
LIN {X 0,Y 83.896,Z 534.917,A -85,B 0,C 180,E1 -28212.079,E2 -28212.079} C_VEL
LIN {X 0,Y 92.428,Z 529.373,A -85,B 0,C 180,E1 -28219.496,E2 -28219.496} C_VEL
LIN {X 0,Y 102.227,Z 522.334,A -85,B 0,C 180,E1 -28225.585,E2 -28225.585} C_VEL
LIN {X 0,Y 112.878,Z 513.583,A -85,B 0,C 180,E1 -28230.65,E2 -28230.65} C_VEL
LIN {X 0,Y 122.903,Z 504.3,A -85,B 0,C 180,E1 -28234.239,E2 -28234.239} C_VEL
LIN {X 0,Y 131.81,Z 494.87,A -85,B 0,C 180,E1 -28236.887,E2 -28236.887} C_VEL
LIN {X 0,Y 140.097,Z 484.879,A -85,B 0,C 180,E1 -28238.887,E2 -28238.887} C_VEL
LIN {X 0,Y 143.173,Z 480.505,A -85,B 0,C 180,E1 -28239.91,E2 -28239.91} C_VEL
LIN {X 0,Y 147.222,Z 473.261,A -85,B 0,C 180,E1 -28242.064,E2 -28242.064} C_VEL
LIN {X 0,Y 151.091,Z 465.702,A -85,B 0,C 180,E1 -28244.005,E2 -28244.005} C_VEL
LIN {X 0,Y 153.773,Z 460.776,A -85,B 0,C 180,E1 -28244.708,E2 -28244.708} C_VEL
LIN {X 0,Y 160.444,Z 447.97,A -85,B 0,C 180,E1 -28245.726,E2 -28245.726} C_VEL
LIN {X 0,Y 166.22,Z 434.426,A -85,B 0,C 180,E1 -28246.519,E2 -28246.519} C_VEL
LIN {X 0,Y 171.189,Z 419.411,A -85,B 0,C 180,E1 -28247.164,E2 -28247.164} C_VEL
LIN {X 0,Y 174.769,Z 404.478,A -85,B 0,C 180,E1 -28247.609,E2 -28247.609} C_VEL
LIN {X 0,Y 177.204,Z 388.13,A -85,B 0,C 180,E1 -28247.975,E2 -28247.975} C_VEL
LIN {X 0,Y 178.798,Z 373.743,A -85,B 0,C 180,E1 -28248.296,E2 -28248.296} C_VEL
LIN {X 0,Y 177.379,Z 369.659,A -85,B 0,C 180,E1 -28251.742,E2 -28251.742} C_VEL
LIN {X 0,Y 176.741,Z 367.592,A -85,B 0,C 180,E1 -28253.98,E2 -28253.98} C_VEL
LIN {X 0,Y 176.117,Z 364.535,A -85,B 0,C 180,E1 -28258.882,E2 -28258.882} C_VEL
LIN {X 0,Y 176.111,Z 364.509,A -85,B 0,C 180,E1 -28261.429,E2 -28261.429} C_VEL
LIN {X 0,Y 176.945,Z 368.304,A -85,B 0,C 180,E1 -28267.274,E2 -28267.274} C_VEL
LIN {X 0,Y 178.083,Z 371.716,A -85,B 0,C 180,E1 -28270.569,E2 -28270.569} C_VEL
LIN {X 0,Y 178.783,Z 373.751,A -85,B 0,C 180,E1 -28272.126,E2 -28272.126} C_VEL
LIN {X 0,Y 175.772,Z 397.978,A -85,B 0,C 180,E1 -28272.649,E2 -28272.649} C_VEL
LIN {X 0,Y 172.525,Z 413.31,A -85,B 0,C 180,E1 -28273.138,E2 -28273.138} C_VEL
LIN {X 0,Y 168.234,Z 427.606,A -85,B 0,C 180,E1 -28273.773,E2 -28273.773} C_VEL
LIN {X 0,Y 162.536,Z 442.093,A -85,B 0,C 180,E1 -28274.656,E2 -28274.656} C_VEL
LIN {X 0,Y 155.885,Z 455.687,A -85,B 0,C 180,E1 -28275.816,E2 -28275.816} C_VEL
LIN {X 0,Y 148.143,Z 468.727,A -85,B 0,C 180,E1 -28277.308,E2 -28277.308} C_VEL
LIN {X 0,Y 139.423,Z 480.923,A -85,B 0,C 180,E1 -28279.069,E2 -28279.069} C_VEL
LIN {X 0,Y 130.101,Z 492.033,A -85,B 0,C 180,E1 -28281.28,E2 -28281.28} C_VEL
LIN {X 0,Y 119.543,Z 502.743,A -85,B 0,C 180,E1 -28284.211,E2 -28284.211} C_VEL
LIN {X 0,Y 109.386,Z 511.759,A -85,B 0,C 180,E1 -28287.944,E2 -28287.944} C_VEL
LIN {X 0,Y 99.633,Z 519.174,A -85,B 0,C 180,E1 -28292.173,E2 -28292.173} C_VEL
LIN {X 0,Y 89.287,Z 526.095,A -85,B 0,C 180,E1 -28298.084,E2 -28298.084} C_VEL
LIN {X 0,Y 80.115,Z 531.524,A -85,B 0,C 180,E1 -28305.43,E2 -28305.43} C_VEL
LIN {X 0,Y 72.484,Z 535.612,A -85,B 0,C 180,E1 -28314.427,E2 -28314.427} C_VEL
LIN {X 0,Y 66.876,Z 538.471,A -85,B 0,C 180,E1 -28325.143,E2 -28325.143} C_VEL
LIN {X 0,Y 63.595,Z 540.179,A -85,B 0,C 180,E1 -28337.231,E2 -28337.231} C_VEL
LIN {X 0,Y 62.699,Z 540.766,A -85,B 0,C 180,E1 -28350,E2 -28350} C_VEL
LIN {X 0,Y 63.593,Z 540.208,A -85,B 0,C 180,E1 -28362.769,E2 -28362.769} C_VEL
LIN {X 0,Y 66.826,Z 538.539,A -85,B 0,C 180,E1 -28374.876,E2 -28374.876} C_VEL
LIN {X 0,Y 72.458,Z 535.712,A -85,B 0,C 180,E1 -28385.588,E2 -28385.588} C_VEL
LIN {X 0,Y 80.118,Z 531.655,A -85,B 0,C 180,E1 -28394.568,E2 -28394.568} C_VEL
LIN {X 0,Y 89.258,Z 526.27,A -85,B 0,C 180,E1 -28401.939,E2 -28401.939} C_VEL
LIN {X 0,Y 99.582,Z 519.4,A -85,B 0,C 180,E1 -28407.874,E2 -28407.874} C_VEL
LIN {X 0,Y 109.322,Z 512.012,A -85,B 0,C 180,E1 -28412.12,E2 -28412.12} C_VEL
LIN {X 0,Y 119.406,Z 503.111,A -85,B 0,C 180,E1 -28415.817,E2 -28415.817} C_VEL
LIN {X 0,Y 128.502,Z 494.013,A -85,B 0,C 180,E1 -28418.394,E2 -28418.394} C_VEL
LIN {X 0,Y 137.782,Z 483.282,A -85,B 0,C 180,E1 -28420.67,E2 -28420.67} C_VEL
LIN {X 0,Y 146.488,Z 471.558,A -85,B 0,C 180,E1 -28422.462,E2 -28422.462} C_VEL
LIN {X 0,Y 154.678,Z 458.355,A -85,B 0,C 180,E1 -28424.032,E2 -28424.032} C_VEL
LIN {X 0,Y 160.872,Z 446.372,A -85,B 0,C 180,E1 -28425.138,E2 -28425.138} C_VEL
LIN {X 0,Y 166.556,Z 433.063,A -85,B 0,C 180,E1 -28426.044,E2 -28426.044} C_VEL
LIN {X 0,Y 171.454,Z 418.384,A -85,B 0,C 180,E1 -28426.781,E2 -28426.781} C_VEL
LIN {X 0,Y 174.993,Z 403.954,A -85,B 0,C 180,E1 -28427.298,E2 -28427.298} C_VEL
LIN {X 0,Y 177.503,Z 387.97,A -85,B 0,C 180,E1 -28427.68,E2 -28427.68} C_VEL
LIN {X 0,Y 179.042,Z 373.935,A -85,B 0,C 180,E1 -28428.017,E2 -28428.017} C_VEL
LIN {X 0,Y 177.706,Z 370.01,A -85,B 0,C 180,E1 -28431.285,E2 -28431.285} C_VEL
LIN {X 0,Y 176.942,Z 367.616,A -85,B 0,C 180,E1 -28434.006,E2 -28434.006} C_VEL
LIN {X 0,Y 176.416,Z 364.504,A -85,B 0,C 180,E1 -28439.429,E2 -28439.429} C_VEL
LIN {X 0,Y 176.417,Z 364.612,A -85,B 0,C 180,E1 -28440.642,E2 -28440.642} C_VEL
LIN {X 0,Y 177.205,Z 368.401,A -85,B 0,C 180,E1 -28446.69,E2 -28446.69} C_VEL
LIN {X 0,Y 178.212,Z 371.439,A -85,B 0,C 180,E1 -28449.719,E2 -28449.719} C_VEL
LIN {X 0,Y 179.073,Z 373.964,A -85,B 0,C 180,E1 -28451.683,E2 -28451.683} C_VEL
LIN {X 0,Y 175.967,Z 399.514,A -85,B 0,C 180,E1 -28452.249,E2 -28452.249} C_VEL
LIN {X 0,Y 172.645,Z 415.126,A -85,B 0,C 180,E1 -28452.659,E2 -28452.659} C_VEL
LIN {X 0,Y 168.309,Z 429.563,A -85,B 0,C 180,E1 -28453.239,E2 -28453.239} C_VEL
LIN {X 0,Y 162.917,Z 443.271,A -85,B 0,C 180,E1 -28453.93,E2 -28453.93} C_VEL
LIN {X 0,Y 156.354,Z 456.707,A -85,B 0,C 180,E1 -28454.898,E2 -28454.898} C_VEL
LIN {X 0,Y 148.24,Z 470.393,A -85,B 0,C 180,E1 -28456.256,E2 -28456.256} C_VEL
LIN {X 0,Y 138.647,Z 483.802,A -85,B 0,C 180,E1 -28458.119,E2 -28458.119} C_VEL
LIN {X 0,Y 129.188,Z 494.954,A -85,B 0,C 180,E1 -28460.216,E2 -28460.216} C_VEL
LIN {X 0,Y 119.976,Z 504.349,A -85,B 0,C 180,E1 -28462.693,E2 -28462.693} C_VEL
LIN {X 0,Y 109.58,Z 513.593,A -85,B 0,C 180,E1 -28466.12,E2 -28466.12} C_VEL
LIN {X 0,Y 99.703,Z 521.29,A -85,B 0,C 180,E1 -28470.291,E2 -28470.291} C_VEL
LIN {X 0,Y 90.469,Z 527.678,A -85,B 0,C 180,E1 -28475.347,E2 -28475.347} C_VEL
LIN {X 0,Y 80.912,Z 533.557,A -85,B 0,C 180,E1 -28482.414,E2 -28482.414} C_VEL
LIN {X 0,Y 74.737,Z 537.062,A -85,B 0,C 180,E1 -28488.835,E2 -28488.835} C_VEL
LIN {X 0,Y 68.2,Z 540.61,A -85,B 0,C 180,E1 -28498.987,E2 -28498.987} C_VEL
LIN {X 0,Y 63.989,Z 542.955,A -85,B 0,C 180,E1 -28510.762,E2 -28510.762} C_VEL
LIN {X 0,Y 62.447,Z 544.147,A -85,B 0,C 180,E1 -28523.538,E2 -28523.538} C_VEL
LIN {X 0,Y 62.555,Z 544.31,A -85,B 0,C 180,E1 -28530,E2 -28530} C_VEL
LIN {X 0,Y 62.88,Z 543.671,A -85,B 0,C 180,E1 -28542.917,E2 -28542.917} C_VEL
LIN {X 0,Y 65.702,Z 541.875,A -85,B 0,C 180,E1 -28555.332,E2 -28555.332} C_VEL
LIN {X 0,Y 71.158,Z 538.913,A -85,B 0,C 180,E1 -28566.34,E2 -28566.34} C_VEL
LIN {X 0,Y 78.724,Z 534.713,A -85,B 0,C 180,E1 -28575.576,E2 -28575.576} C_VEL
LIN {X 0,Y 87.935,Z 529.168,A -85,B 0,C 180,E1 -28583.055,E2 -28583.055} C_VEL
LIN {X 0,Y 98.33,Z 522.128,A -85,B 0,C 180,E1 -28589.056,E2 -28589.056} C_VEL
LIN {X 0,Y 108.095,Z 514.607,A -85,B 0,C 180,E1 -28593.373,E2 -28593.373} C_VEL
LIN {X 0,Y 118.455,Z 505.55,A -85,B 0,C 180,E1 -28596.868,E2 -28596.868} C_VEL
LIN {X 0,Y 129.183,Z 494.666,A -85,B 0,C 180,E1 -28599.791,E2 -28599.791} C_VEL
LIN {X 0,Y 138.658,Z 483.471,A -85,B 0,C 180,E1 -28601.867,E2 -28601.867} C_VEL
LIN {X 0,Y 147.423,Z 471.195,A -85,B 0,C 180,E1 -28603.614,E2 -28603.614} C_VEL
LIN {X 0,Y 153.773,Z 460.776,A -85,B 0,C 180,E1 -28604.708,E2 -28604.708} C_VEL
LIN {X 0,Y 156.378,Z 455.808,A -85,B 0,C 180,E1 -28605.358,E2 -28605.358} C_VEL
LIN {X 0,Y 159.824,Z 447.598,A -85,B 0,C 180,E1 -28606.956,E2 -28606.956} C_VEL
LIN {X 0,Y 162.909,Z 439.171,A -85,B 0,C 180,E1 -28608.447,E2 -28608.447} C_VEL
LIN {X 0,Y 164.867,Z 433.789,A -85,B 0,C 180,E1 -28608.944,E2 -28608.944} C_VEL
LIN {X 0,Y 169.755,Z 419.201,A -85,B 0,C 180,E1 -28609.498,E2 -28609.498} C_VEL
LIN {X 0,Y 173.293,Z 404.772,A -85,B 0,C 180,E1 -28609.887,E2 -28609.887} C_VEL
LIN {X 0,Y 175.818,Z 388.275,A -85,B 0,C 180,E1 -28610.235,E2 -28610.235} C_VEL
LIN {X 0,Y 176.927,Z 378.505,A -85,B 0,C 180,E1 -28610.437,E2 -28610.437} C_VEL
LIN {X 0,Y 175.785,Z 374.579,A -85,B 0,C 180,E1 -28614.264,E2 -28614.264} C_VEL
LIN {X 0,Y 175.232,Z 371.486,A -85,B 0,C 180,E1 -28619.438,E2 -28619.438} C_VEL
LIN {X 0,Y 175.233,Z 371.669,A -85,B 0,C 180,E1 -28621.437,E2 -28621.437} C_VEL
LIN {X 0,Y 175.905,Z 375.136,A -85,B 0,C 180,E1 -28626.74,E2 -28626.74} C_VEL
LIN {X 0,Y 176.918,Z 378.504,A -85,B 0,C 180,E1 -28629.988,E2 -28629.988} C_VEL
LIN {X 0,Y 174.186,Z 399.156,A -85,B 0,C 180,E1 -28630.409,E2 -28630.409} C_VEL
LIN {X 0,Y 170.834,Z 414.311,A -85,B 0,C 180,E1 -28630.849,E2 -28630.849} C_VEL
LIN {X 0,Y 166.252,Z 429.006,A -85,B 0,C 180,E1 -28631.47,E2 -28631.47} C_VEL
LIN {X 0,Y 160.888,Z 442.299,A -85,B 0,C 180,E1 -28632.211,E2 -28632.211} C_VEL
LIN {X 0,Y 154.096,Z 455.893,A -85,B 0,C 180,E1 -28633.266,E2 -28633.266} C_VEL
LIN {X 0,Y 146.188,Z 468.932,A -85,B 0,C 180,E1 -28634.649,E2 -28634.649} C_VEL
LIN {X 0,Y 137.27,Z 481.126,A -85,B 0,C 180,E1 -28636.271,E2 -28636.271} C_VEL
LIN {X 0,Y 127.699,Z 492.236,A -85,B 0,C 180,E1 -28638.315,E2 -28638.315} C_VEL
LIN {X 0,Y 118.156,Z 501.687,A -85,B 0,C 180,E1 -28640.659,E2 -28640.659} C_VEL
LIN {X 0,Y 107.728,Z 510.749,A -85,B 0,C 180,E1 -28644.033,E2 -28644.033} C_VEL
LIN {X 0,Y 97.45,Z 518.377,A -85,B 0,C 180,E1 -28647.94,E2 -28647.94} C_VEL
LIN {X 0,Y 87.734,Z 524.699,A -85,B 0,C 180,E1 -28652.744,E2 -28652.744} C_VEL
LIN {X 0,Y 78.664,Z 529.924,A -85,B 0,C 180,E1 -28658.712,E2 -28658.712} C_VEL
LIN {X 0,Y 70.847,Z 533.928,A -85,B 0,C 180,E1 -28666.022,E2 -28666.022} C_VEL
LIN {X 0,Y 63.325,Z 537.393,A -85,B 0,C 180,E1 -28676.296,E2 -28676.296} C_VEL
LIN {X 0,Y 58.245,Z 539.667,A -85,B 0,C 180,E1 -28688.778,E2 -28688.778} C_VEL
LIN {X 0,Y 55.825,Z 540.816,A -85,B 0,C 180,E1 -28702.768,E2 -28702.768} C_VEL
LIN {X 0,Y 55.608,Z 540.967,A -85,B 0,C 180,E1 -28710,E2 -28710} C_VEL
LIN {X 0,Y 56.674,Z 540.409,A -85,B 0,C 180,E1 -28724.36,E2 -28724.36} C_VEL
LIN {X 0,Y 60.424,Z 538.741,A -85,B 0,C 180,E1 -28737.725,E2 -28737.725} C_VEL
LIN {X 0,Y 66.801,Z 535.913,A -85,B 0,C 180,E1 -28749.141,E2 -28749.141} C_VEL
LIN {X 0,Y 75.202,Z 531.856,A -85,B 0,C 180,E1 -28758.385,E2 -28758.385} C_VEL
LIN {X 0,Y 85.041,Z 526.471,A -85,B 0,C 180,E1 -28765.731,E2 -28765.731} C_VEL
LIN {X 0,Y 95.972,Z 519.6,A -85,B 0,C 180,E1 -28771.49,E2 -28771.49} C_VEL
LIN {X 0,Y 106.177,Z 512.212,A -85,B 0,C 180,E1 -28775.52,E2 -28775.52} C_VEL
LIN {X 0,Y 116.676,Z 503.31,A -85,B 0,C 180,E1 -28779.001,E2 -28779.001} C_VEL
LIN {X 0,Y 126.062,Z 494.211,A -85,B 0,C 180,E1 -28781.394,E2 -28781.394} C_VEL
LIN {X 0,Y 135.598,Z 483.48,A -85,B 0,C 180,E1 -28783.501,E2 -28783.501} C_VEL
LIN {X 0,Y 144.508,Z 471.755,A -85,B 0,C 180,E1 -28785.145,E2 -28785.145} C_VEL
LIN {X 0,Y 152.871,Z 458.552,A -85,B 0,C 180,E1 -28786.601,E2 -28786.601} C_VEL
LIN {X 0,Y 160.03,Z 444.805,A -85,B 0,C 180,E1 -28787.721,E2 -28787.721} C_VEL
LIN {X 0,Y 165.821,Z 431.002,A -85,B 0,C 180,E1 -28788.546,E2 -28788.546} C_VEL
LIN {X 0,Y 170.796,Z 415.533,A -85,B 0,C 180,E1 -28789.234,E2 -28789.234} C_VEL
LIN {X 0,Y 174.265,Z 400.398,A -85,B 0,C 180,E1 -28789.676,E2 -28789.676} C_VEL
LIN {X 0,Y 176.989,Z 380.724,A -85,B 0,C 180,E1 -28790.052,E2 -28790.052} C_VEL
LIN {X 0,Y 177.184,Z 378.682,A -85,B 0,C 180,E1 -28790.163,E2 -28790.163} C_VEL
LIN {X 0,Y 176.065,Z 374.795,A -85,B 0,C 180,E1 -28793.976,E2 -28793.976} C_VEL
LIN {X 0,Y 175.549,Z 371.566,A -85,B 0,C 180,E1 -28799.426,E2 -28799.426} C_VEL
LIN {X 0,Y 175.54,Z 371.692,A -85,B 0,C 180,E1 -28800.43,E2 -28800.43} C_VEL
LIN {X 0,Y 176.204,Z 375.352,A -85,B 0,C 180,E1 -28806.297,E2 -28806.297} C_VEL
LIN {X 0,Y 177.208,Z 378.714,A -85,B 0,C 180,E1 -28809.537,E2 -28809.537} C_VEL
LIN {X 0,Y 174.454,Z 400.122,A -85,B 0,C 180,E1 -28809.992,E2 -28809.992} C_VEL
LIN {X 0,Y 171.098,Z 415.411,A -85,B 0,C 180,E1 -28810.355,E2 -28810.355} C_VEL
LIN {X 0,Y 166.408,Z 430.501,A -85,B 0,C 180,E1 -28810.917,E2 -28810.917} C_VEL
LIN {X 0,Y 160.513,Z 444.862,A -85,B 0,C 180,E1 -28811.577,E2 -28811.577} C_VEL
LIN {X 0,Y 153.847,Z 458.001,A -85,B 0,C 180,E1 -28812.465,E2 -28812.465} C_VEL
LIN {X 0,Y 145.582,Z 471.396,A -85,B 0,C 180,E1 -28813.708,E2 -28813.708} C_VEL
LIN {X 0,Y 136.593,Z 483.603,A -85,B 0,C 180,E1 -28815.269,E2 -28815.269} C_VEL
LIN {X 0,Y 126.906,Z 494.755,A -85,B 0,C 180,E1 -28817.201,E2 -28817.201} C_VEL
LIN {X 0,Y 117.398,Z 504.149,A -85,B 0,C 180,E1 -28819.465,E2 -28819.465} C_VEL
LIN {X 0,Y 106.611,Z 513.392,A -85,B 0,C 180,E1 -28822.649,E2 -28822.649} C_VEL
LIN {X 0,Y 96.293,Z 521.089,A -85,B 0,C 180,E1 -28826.613,E2 -28826.613} C_VEL
LIN {X 0,Y 86.517,Z 527.476,A -85,B 0,C 180,E1 -28831.469,E2 -28831.469} C_VEL
LIN {X 0,Y 76.263,Z 533.355,A -85,B 0,C 180,E1 -28838.437,E2 -28838.437} C_VEL
LIN {X 0,Y 69.051,Z 537.087,A -85,B 0,C 180,E1 -28845.434,E2 -28845.434} C_VEL
LIN {X 0,Y 62.165,Z 540.408,A -85,B 0,C 180,E1 -28855.58,E2 -28855.58} C_VEL
LIN {X 0,Y 57.277,Z 542.752,A -85,B 0,C 180,E1 -28868.402,E2 -28868.402} C_VEL
LIN {X 0,Y 55.366,Z 543.945,A -85,B 0,C 180,E1 -28882.708,E2 -28882.708} C_VEL
LIN {X 0,Y 55.463,Z 544.11,A -85,B 0,C 180,E1 -28890,E2 -28890} C_VEL
LIN {X 0,Y 55.953,Z 543.469,A -85,B 0,C 180,E1 -28904.549,E2 -28904.549} C_VEL
LIN {X 0,Y 59.312,Z 541.672,A -85,B 0,C 180,E1 -28918.292,E2 -28918.292} C_VEL
LIN {X 0,Y 65.52,Z 538.709,A -85,B 0,C 180,E1 -28930.059,E2 -28930.059} C_VEL
LIN {X 0,Y 73.872,Z 534.509,A -85,B 0,C 180,E1 -28939.56,E2 -28939.56} C_VEL
LIN {X 0,Y 83.82,Z 528.964,A -85,B 0,C 180,E1 -28946.976,E2 -28946.976} C_VEL
LIN {X 0,Y 94.839,Z 521.924,A -85,B 0,C 180,E1 -28952.778,E2 -28952.778} C_VEL
LIN {X 0,Y 105.077,Z 514.401,A -85,B 0,C 180,E1 -28956.873,E2 -28956.873} C_VEL
LIN {X 0,Y 115.837,Z 505.346,A -85,B 0,C 180,E1 -28960.116,E2 -28960.116} C_VEL
LIN {X 0,Y 125.288,Z 496.103,A -85,B 0,C 180,E1 -28962.476,E2 -28962.476} C_VEL
LIN {X 0,Y 134.987,Z 485.224,A -85,B 0,C 180,E1 -28964.402,E2 -28964.402} C_VEL
LIN {X 0,Y 143.603,Z 473.82,A -85,B 0,C 180,E1 -28965.977,E2 -28965.977} C_VEL
LIN {X 0,Y 151.658,Z 461.246,A -85,B 0,C 180,E1 -28967.242,E2 -28967.242} C_VEL
LIN {X 0,Y 158.84,Z 447.763,A -85,B 0,C 180,E1 -28968.214,E2 -28968.214} C_VEL
LIN {X 0,Y 164.867,Z 433.789,A -85,B 0,C 180,E1 -28968.944,E2 -28968.944} C_VEL
LIN {X 0,Y 166.758,Z 428.326,A -85,B 0,C 180,E1 -28969.399,E2 -28969.399} C_VEL
LIN {X 0,Y 170.648,Z 412.247,A -85,B 0,C 180,E1 -28971.678,E2 -28971.678} C_VEL
LIN {X 0,Y 171.783,Z 406.624,A -85,B 0,C 180,E1 -28972.146,E2 -28972.146} C_VEL
LIN {X 0,Y 172.159,Z 404.703,A -85,B 0,C 180,E1 -28972.212,E2 -28972.212} C_VEL
LIN {X 0,Y 174.598,Z 389.41,A -85,B 0,C 180,E1 -28972.499,E2 -28972.499} C_VEL
LIN {X 0,Y 175.272,Z 383.447,A -85,B 0,C 180,E1 -28972.657,E2 -28972.657} C_VEL
LIN {X 0,Y 174.711,Z 381.285,A -85,B 0,C 180,E1 -28975.097,E2 -28975.097} C_VEL
LIN {X 0,Y 174.361,Z 378.456,A -85,B 0,C 180,E1 -28980,E2 -28980} C_VEL
LIN {X 0,Y 174.337,Z 379.1,A -85,B 0,C 180,E1 -28981.678,E2 -28981.678} C_VEL
LIN {X 0,Y 174.872,Z 381.94,A -85,B 0,C 180,E1 -28986.165,E2 -28986.165} C_VEL
LIN {X 0,Y 175.272,Z 383.495,A -85,B 0,C 180,E1 -28987.8,E2 -28987.8} C_VEL
LIN {X 0,Y 172.634,Z 401.585,A -85,B 0,C 180,E1 -28988.143,E2 -28988.143} C_VEL
LIN {X 0,Y 169.051,Z 416.661,A -85,B 0,C 180,E1 -28988.57,E2 -28988.57} C_VEL
LIN {X 0,Y 164.121,Z 431.514,A -85,B 0,C 180,E1 -28989.145,E2 -28989.145} C_VEL
LIN {X 0,Y 157.857,Z 446.027,A -85,B 0,C 180,E1 -28989.933,E2 -28989.933} C_VEL
LIN {X 0,Y 150.962,Z 458.947,A -85,B 0,C 180,E1 -28990.931,E2 -28990.931} C_VEL
LIN {X 0,Y 142.894,Z 471.474,A -85,B 0,C 180,E1 -28992.179,E2 -28992.179} C_VEL
LIN {X 0,Y 133.802,Z 483.274,A -85,B 0,C 180,E1 -28993.664,E2 -28993.664} C_VEL
LIN {X 0,Y 124.011,Z 494.069,A -85,B 0,C 180,E1 -28995.547,E2 -28995.547} C_VEL
LIN {X 0,Y 114.354,Z 503.227,A -85,B 0,C 180,E1 -28997.721,E2 -28997.721} C_VEL
LIN {X 0,Y 103.485,Z 512.165,A -85,B 0,C 180,E1 -29000.967,E2 -29000.967} C_VEL
LIN {X 0,Y 92.829,Z 519.58,A -85,B 0,C 180,E1 -29004.703,E2 -29004.703} C_VEL
LIN {X 0,Y 81.274,Z 526.501,A -85,B 0,C 180,E1 -29010.15,E2 -29010.15} C_VEL
LIN {X 0,Y 70.666,Z 531.93,A -85,B 0,C 180,E1 -29017.286,E2 -29017.286} C_VEL
LIN {X 0,Y 61.469,Z 536.016,A -85,B 0,C 180,E1 -29026.687,E2 -29026.687} C_VEL
LIN {X 0,Y 54.256,Z 538.876,A -85,B 0,C 180,E1 -29038.793,E2 -29038.793} C_VEL
LIN {X 0,Y 49.83,Z 540.581,A -85,B 0,C 180,E1 -29053.616,E2 -29053.616} C_VEL
LIN {X 0,Y 48.508,Z 541.168,A -85,B 0,C 180,E1 -29070,E2 -29070} C_VEL
LIN {X 0,Y 49.823,Z 540.609,A -85,B 0,C 180,E1 -29086.386,E2 -29086.386} C_VEL
LIN {X 0,Y 54.215,Z 538.942,A -85,B 0,C 180,E1 -29101.233,E2 -29101.233} C_VEL
LIN {X 0,Y 61.449,Z 536.113,A -85,B 0,C 180,E1 -29113.331,E2 -29113.331} C_VEL
LIN {X 0,Y 70.667,Z 532.056,A -85,B 0,C 180,E1 -29122.712,E2 -29122.712} C_VEL
LIN {X 0,Y 81.232,Z 526.672,A -85,B 0,C 180,E1 -29129.9,E2 -29129.9} C_VEL
LIN {X 0,Y 92.775,Z 519.801,A -85,B 0,C 180,E1 -29135.37,E2 -29135.37} C_VEL
LIN {X 0,Y 103.427,Z 512.412,A -85,B 0,C 180,E1 -29139.117,E2 -29139.117} C_VEL
LIN {X 0,Y 114.002,Z 503.776,A -85,B 0,C 180,E1 -29142.259,E2 -29142.259} C_VEL
LIN {X 0,Y 123.983,Z 494.409,A -85,B 0,C 180,E1 -29144.499,E2 -29144.499} C_VEL
LIN {X 0,Y 133.757,Z 483.677,A -85,B 0,C 180,E1 -29146.416,E2 -29146.416} C_VEL
LIN {X 0,Y 142.854,Z 471.952,A -85,B 0,C 180,E1 -29147.896,E2 -29147.896} C_VEL
LIN {X 0,Y 151.309,Z 458.867,A -85,B 0,C 180,E1 -29149.214,E2 -29149.214} C_VEL
LIN {X 0,Y 158.671,Z 445.001,A -85,B 0,C 180,E1 -29150.228,E2 -29150.228} C_VEL
LIN {X 0,Y 164.913,Z 430.256,A -85,B 0,C 180,E1 -29151.005,E2 -29151.005} C_VEL
LIN {X 0,Y 169.784,Z 415.123,A -85,B 0,C 180,E1 -29151.601,E2 -29151.601} C_VEL
LIN {X 0,Y 173.326,Z 399.54,A -85,B 0,C 180,E1 -29152.015,E2 -29152.015} C_VEL
LIN {X 0,Y 175.559,Z 383.674,A -85,B 0,C 180,E1 -29152.326,E2 -29152.326} C_VEL
LIN {X 0,Y 174.943,Z 381.308,A -85,B 0,C 180,E1 -29155.103,E2 -29155.103} C_VEL
LIN {X 0,Y 174.674,Z 378.693,A -85,B 0,C 180,E1 -29159.423,E2 -29159.423} C_VEL
LIN {X 0,Y 174.661,Z 378.817,A -85,B 0,C 180,E1 -29160.288,E2 -29160.288} C_VEL
LIN {X 0,Y 175.176,Z 382.215,A -85,B 0,C 180,E1 -29165.756,E2 -29165.756} C_VEL
LIN {X 0,Y 175.569,Z 383.636,A -85,B 0,C 180,E1 -29167.334,E2 -29167.334} C_VEL
LIN {X 0,Y 173.106,Z 401.324,A -85,B 0,C 180,E1 -29167.711,E2 -29167.711} C_VEL
LIN {X 0,Y 169.577,Z 416.598,A -85,B 0,C 180,E1 -29168.03,E2 -29168.03} C_VEL
LIN {X 0,Y 164.737,Z 431.562,A -85,B 0,C 180,E1 -29168.542,E2 -29168.542} C_VEL
LIN {X 0,Y 158.391,Z 446.435,A -85,B 0,C 180,E1 -29169.164,E2 -29169.164} C_VEL
LIN {X 0,Y 150.779,Z 460.66,A -85,B 0,C 180,E1 -29170.056,E2 -29170.056} C_VEL
LIN {X 0,Y 142.312,Z 473.665,A -85,B 0,C 180,E1 -29171.215,E2 -29171.215} C_VEL
LIN {X 0,Y 133.242,Z 485.365,A -85,B 0,C 180,E1 -29172.637,E2 -29172.637} C_VEL
LIN {X 0,Y 123.337,Z 496.19,A -85,B 0,C 180,E1 -29174.38,E2 -29174.38} C_VEL
LIN {X 0,Y 113.605,Z 505.38,A -85,B 0,C 180,E1 -29176.492,E2 -29176.492} C_VEL
LIN {X 0,Y 102.502,Z 514.405,A -85,B 0,C 180,E1 -29179.484,E2 -29179.484} C_VEL
LIN {X 0,Y 91.792,Z 521.903,A -85,B 0,C 180,E1 -29183.256,E2 -29183.256} C_VEL
LIN {X 0,Y 80.14,Z 528.9,A -85,B 0,C 180,E1 -29188.724,E2 -29188.724} C_VEL
LIN {X 0,Y 69.468,Z 534.41,A -85,B 0,C 180,E1 -29195.969,E2 -29195.969} C_VEL
LIN {X 0,Y 60.249,Z 538.586,A -85,B 0,C 180,E1 -29205.583,E2 -29205.583} C_VEL
LIN {X 0,Y 53.142,Z 541.523,A -85,B 0,C 180,E1 -29218.063,E2 -29218.063} C_VEL
LIN {X 0,Y 49.067,Z 543.289,A -85,B 0,C 180,E1 -29233.354,E2 -29233.354} C_VEL
LIN {X 0,Y 48.355,Z 543.908,A -85,B 0,C 180,E1 -29250,E2 -29250} C_VEL
LIN {X 0,Y 49.063,Z 543.266,A -85,B 0,C 180,E1 -29266.648,E2 -29266.648} C_VEL
LIN {X 0,Y 53.123,Z 541.47,A -85,B 0,C 180,E1 -29281.95,E2 -29281.95} C_VEL
LIN {X 0,Y 60.195,Z 538.505,A -85,B 0,C 180,E1 -29294.468,E2 -29294.468} C_VEL
LIN {X 0,Y 69.445,Z 534.306,A -85,B 0,C 180,E1 -29304.057,E2 -29304.057} C_VEL
LIN {X 0,Y 80.137,Z 528.76,A -85,B 0,C 180,E1 -29311.279,E2 -29311.279} C_VEL
LIN {X 0,Y 91.786,Z 521.719,A -85,B 0,C 180,E1 -29316.753,E2 -29316.753} C_VEL
LIN {X 0,Y 102.48,Z 514.197,A -85,B 0,C 180,E1 -29320.552,E2 -29320.552} C_VEL
LIN {X 0,Y 113.6,Z 505.141,A -85,B 0,C 180,E1 -29323.518,E2 -29323.518} C_VEL
LIN {X 0,Y 123.334,Z 495.899,A -85,B 0,C 180,E1 -29325.627,E2 -29325.627} C_VEL
LIN {X 0,Y 133.245,Z 485.019,A -85,B 0,C 180,E1 -29327.36,E2 -29327.36} C_VEL
LIN {X 0,Y 141.875,Z 473.854,A -85,B 0,C 180,E1 -29328.742,E2 -29328.742} C_VEL
LIN {X 0,Y 149.932,Z 461.576,A -85,B 0,C 180,E1 -29329.847,E2 -29329.847} C_VEL
LIN {X 0,Y 157.538,Z 447.555,A -85,B 0,C 180,E1 -29330.753,E2 -29330.753} C_VEL
LIN {X 0,Y 163.883,Z 432.968,A -85,B 0,C 180,E1 -29331.412,E2 -29331.412} C_VEL
LIN {X 0,Y 168.896,Z 417.94,A -85,B 0,C 180,E1 -29331.905,E2 -29331.905} C_VEL
LIN {X 0,Y 172.159,Z 404.703,A -85,B 0,C 180,E1 -29332.212,E2 -29332.212} C_VEL
LIN {X 0,Y 172.882,Z 400.513,A -85,B 0,C 180,E1 -29332.466,E2 -29332.466} C_VEL
LIN {X 0,Y 173.362,Z 396.538,A -85,B 0,C 180,E1 -29333.016,E2 -29333.016} C_VEL
LIN {X 0,Y 173.662,Z 391.909,A -85,B 0,C 180,E1 -29334.106,E2 -29334.106} C_VEL
LIN {X 0,Y 173.712,Z 389.245,A -85,B 0,C 180,E1 -29335.174,E2 -29335.174} C_VEL
LIN {X 0,Y 173.602,Z 387.703,A -85,B 0,C 180,E1 -29336.439,E2 -29336.439} C_VEL
LIN {X 0,Y 173.492,Z 385.53,A -85,B 0,C 180,E1 -29340,E2 -29340} C_VEL
LIN {X 0,Y 173.451,Z 386.354,A -85,B 0,C 180,E1 -29341.742,E2 -29341.742} C_VEL
LIN {X 0,Y 173.854,Z 388.763,A -85,B 0,C 180,E1 -29345.581,E2 -29345.581} C_VEL
LIN {X 0,Y 171.322,Z 404.215,A -85,B 0,C 180,E1 -29345.866,E2 -29345.866} C_VEL
LIN {X 0,Y 167.268,Z 419.918,A -85,B 0,C 180,E1 -29346.269,E2 -29346.269} C_VEL
LIN {X 0,Y 161.91,Z 434.919,A -85,B 0,C 180,E1 -29346.829,E2 -29346.829} C_VEL
LIN {X 0,Y 155.195,Z 449.446,A -85,B 0,C 180,E1 -29347.56,E2 -29347.56} C_VEL
LIN {X 0,Y 147.477,Z 462.959,A -85,B 0,C 180,E1 -29348.578,E2 -29348.578} C_VEL
LIN {X 0,Y 139.035,Z 475.173,A -85,B 0,C 180,E1 -29349.711,E2 -29349.711} C_VEL
LIN {X 0,Y 128.962,Z 487.333,A -85,B 0,C 180,E1 -29351.211,E2 -29351.211} C_VEL
LIN {X 0,Y 118.975,Z 497.513,A -85,B 0,C 180,E1 -29352.928,E2 -29352.928} C_VEL
LIN {X 0,Y 108.092,Z 506.983,A -85,B 0,C 180,E1 -29355.249,E2 -29355.249} C_VEL
LIN {X 0,Y 97.948,Z 514.592,A -85,B 0,C 180,E1 -29358.067,E2 -29358.067} C_VEL
LIN {X 0,Y 86.989,Z 521.647,A -85,B 0,C 180,E1 -29361.707,E2 -29361.707} C_VEL
LIN {X 0,Y 74.997,Z 528.186,A -85,B 0,C 180,E1 -29367.098,E2 -29367.098} C_VEL
LIN {X 0,Y 63.912,Z 533.285,A -85,B 0,C 180,E1 -29374.441,E2 -29374.441} C_VEL
LIN {X 0,Y 56.484,Z 536.218,A -85,B 0,C 180,E1 -29381.709,E2 -29381.709} C_VEL
LIN {X 0,Y 48.303,Z 539.078,A -85,B 0,C 180,E1 -29394.41,E2 -29394.41} C_VEL
LIN {X 0,Y 43.047,Z 540.783,A -85,B 0,C 180,E1 -29410.942,E2 -29410.942} C_VEL
LIN {X 0,Y 41.426,Z 541.368,A -85,B 0,C 180,E1 -29430,E2 -29430} C_VEL
LIN {X 0,Y 43.039,Z 540.811,A -85,B 0,C 180,E1 -29449.061,E2 -29449.061} C_VEL
LIN {X 0,Y 48.266,Z 539.143,A -85,B 0,C 180,E1 -29465.621,E2 -29465.621} C_VEL
LIN {X 0,Y 56.465,Z 536.314,A -85,B 0,C 180,E1 -29478.312,E2 -29478.312} C_VEL
LIN {X 0,Y 66.589,Z 532.257,A -85,B 0,C 180,E1 -29487.599,E2 -29487.599} C_VEL
LIN {X 0,Y 77.904,Z 526.872,A -85,B 0,C 180,E1 -29494.437,E2 -29494.437} C_VEL
LIN {X 0,Y 90.029,Z 520.002,A -85,B 0,C 180,E1 -29499.512,E2 -29499.512} C_VEL
LIN {X 0,Y 102.692,Z 511.418,A -85,B 0,C 180,E1 -29503.357,E2 -29503.357} C_VEL
LIN {X 0,Y 110.728,Z 505.052,A -85,B 0,C 180,E1 -29505.445,E2 -29505.445} C_VEL
LIN {X 0,Y 120.612,Z 496.227,A -85,B 0,C 180,E1 -29507.419,E2 -29507.419} C_VEL
LIN {X 0,Y 130.59,Z 485.82,A -85,B 0,C 180,E1 -29509.156,E2 -29509.156} C_VEL
LIN {X 0,Y 139.84,Z 474.489,A -85,B 0,C 180,E1 -29510.498,E2 -29510.498} C_VEL
LIN {X 0,Y 148.289,Z 462.177,A -85,B 0,C 180,E1 -29511.619,E2 -29511.619} C_VEL
LIN {X 0,Y 155.918,Z 448.705,A -85,B 0,C 180,E1 -29512.579,E2 -29512.579} C_VEL
LIN {X 0,Y 162.311,Z 434.73,A -85,B 0,C 180,E1 -29513.295,E2 -29513.295} C_VEL
LIN {X 0,Y 167.539,Z 420.058,A -85,B 0,C 180,E1 -29513.842,E2 -29513.842} C_VEL
LIN {X 0,Y 171.382,Z 405.353,A -85,B 0,C 180,E1 -29514.231,E2 -29514.231} C_VEL
LIN {X 0,Y 174.042,Z 389.805,A -85,B 0,C 180,E1 -29514.496,E2 -29514.496} C_VEL
LIN {X 0,Y 174.139,Z 388.966,A -85,B 0,C 180,E1 -29514.572,E2 -29514.572} C_VEL
LIN {X 0,Y 173.79,Z 385.892,A -85,B 0,C 180,E1 -29519.42,E2 -29519.42} C_VEL
LIN {X 0,Y 173.765,Z 386.189,A -85,B 0,C 180,E1 -29520.579,E2 -29520.579} C_VEL
LIN {X 0,Y 174.156,Z 388.986,A -85,B 0,C 180,E1 -29525.141,E2 -29525.141} C_VEL
LIN {X 0,Y 171.5,Z 405.303,A -85,B 0,C 180,E1 -29525.423,E2 -29525.423} C_VEL
LIN {X 0,Y 167.487,Z 420.782,A -85,B 0,C 180,E1 -29525.754,E2 -29525.754} C_VEL
LIN {X 0,Y 162.157,Z 435.73,A -85,B 0,C 180,E1 -29526.225,E2 -29526.225} C_VEL
LIN {X 0,Y 155.702,Z 449.767,A -85,B 0,C 180,E1 -29526.784,E2 -29526.784} C_VEL
LIN {X 0,Y 147.994,Z 463.314,A -85,B 0,C 180,E1 -29527.565,E2 -29527.565} C_VEL
LIN {X 0,Y 139.547,Z 475.618,A -85,B 0,C 180,E1 -29528.572,E2 -29528.572} C_VEL
LIN {X 0,Y 130.184,Z 487.126,A -85,B 0,C 180,E1 -29529.868,E2 -29529.868} C_VEL
LIN {X 0,Y 120.082,Z 497.624,A -85,B 0,C 180,E1 -29531.392,E2 -29531.392} C_VEL
LIN {X 0,Y 108.492,Z 507.902,A -85,B 0,C 180,E1 -29533.673,E2 -29533.673} C_VEL
LIN {X 0,Y 97.115,Z 516.452,A -85,B 0,C 180,E1 -29536.495,E2 -29536.495} C_VEL
LIN {X 0,Y 86.098,Z 523.576,A -85,B 0,C 180,E1 -29540.167,E2 -29540.167} C_VEL
LIN {X 0,Y 73.998,Z 530.189,A -85,B 0,C 180,E1 -29545.545,E2 -29545.545} C_VEL
LIN {X 0,Y 62.831,Z 535.375,A -85,B 0,C 180,E1 -29552.976,E2 -29552.976} C_VEL
LIN {X 0,Y 55.35,Z 538.384,A -85,B 0,C 180,E1 -29560.375,E2 -29560.375} C_VEL
LIN {X 0,Y 47.228,Z 541.322,A -85,B 0,C 180,E1 -29573.471,E2 -29573.471} C_VEL
LIN {X 0,Y 42.273,Z 543.087,A -85,B 0,C 180,E1 -29590.58,E2 -29590.58} C_VEL
LIN {X 0,Y 41.264,Z 543.708,A -85,B 0,C 180,E1 -29610,E2 -29610} C_VEL
LIN {X 0,Y 42.269,Z 543.064,A -85,B 0,C 180,E1 -29629.423,E2 -29629.423} C_VEL
LIN {X 0,Y 47.208,Z 541.267,A -85,B 0,C 180,E1 -29646.547,E2 -29646.547} C_VEL
LIN {X 0,Y 55.301,Z 538.301,A -85,B 0,C 180,E1 -29659.685,E2 -29659.685} C_VEL
LIN {X 0,Y 65.494,Z 534.102,A -85,B 0,C 180,E1 -29669.142,E2 -29669.142} C_VEL
LIN {X 0,Y 76.948,Z 528.556,A -85,B 0,C 180,E1 -29675.968,E2 -29675.968} C_VEL
LIN {X 0,Y 89.2,Z 521.515,A -85,B 0,C 180,E1 -29680.988,E2 -29680.988} C_VEL
LIN {X 0,Y 100.326,Z 513.993,A -85,B 0,C 180,E1 -29684.405,E2 -29684.405} C_VEL
LIN {X 0,Y 111.779,Z 504.936,A -85,B 0,C 180,E1 -29687.039,E2 -29687.039} C_VEL
LIN {X 0,Y 121.758,Z 495.694,A -85,B 0,C 180,E1 -29688.883,E2 -29688.883} C_VEL
LIN {X 0,Y 131.865,Z 484.814,A -85,B 0,C 180,E1 -29690.392,E2 -29690.392} C_VEL
LIN {X 0,Y 141.254,Z 472.817,A -85,B 0,C 180,E1 -29691.673,E2 -29691.673} C_VEL
LIN {X 0,Y 149.697,Z 459.94,A -85,B 0,C 180,E1 -29692.638,E2 -29692.638} C_VEL
LIN {X 0,Y 157.409,Z 445.579,A -85,B 0,C 180,E1 -29693.411,E2 -29693.411} C_VEL
LIN {X 0,Y 163.289,Z 431.934,A -85,B 0,C 180,E1 -29693.906,E2 -29693.906} C_VEL
LIN {X 0,Y 168.462,Z 416.25,A -85,B 0,C 180,E1 -29694.333,E2 -29694.333} C_VEL
LIN {X 0,Y 172.051,Z 400.737,A -85,B 0,C 180,E1 -29694.621,E2 -29694.621} C_VEL
LIN {X 0,Y 173.864,Z 388.729,A -85,B 0,C 180,E1 -29694.845,E2 -29694.845} C_VEL
LIN {X 0,Y 173.602,Z 387.703,A -85,B 0,C 180,E1 -29696.439,E2 -29696.439} C_VEL
LIN {X 0,Y 173.383,Z 387.77,A -85,B 0,C 180,E1 -29697.724,E2 -29697.724} C_VEL
LIN {X 0,Y 173.023,Z 389.492,A -85,B 0,C 180,E1 -29699.378,E2 -29699.378} C_VEL
LIN {X 0,Y 172.508,Z 393.643,A -85,B 0,C 180,E1 -29702.253,E2 -29702.253} C_VEL
LIN {X 0,Y 172.515,Z 394.35,A -85,B 0,C 180,E1 -29703.133,E2 -29703.133} C_VEL
LIN {X 0,Y 172.534,Z 394.409,A -85,B 0,C 180,E1 -29703.309,E2 -29703.309} C_VEL
LIN {X 0,Y 169.656,Z 409.05,A -85,B 0,C 180,E1 -29703.573,E2 -29703.573} C_VEL
LIN {X 0,Y 165.808,Z 422.636,A -85,B 0,C 180,E1 -29703.922,E2 -29703.922} C_VEL
LIN {X 0,Y 160.353,Z 437.108,A -85,B 0,C 180,E1 -29704.389,E2 -29704.389} C_VEL
LIN {X 0,Y 153.59,Z 451.174,A -85,B 0,C 180,E1 -29705.031,E2 -29705.031} C_VEL
LIN {X 0,Y 145.728,Z 464.451,A -85,B 0,C 180,E1 -29705.928,E2 -29705.928} C_VEL
LIN {X 0,Y 137.158,Z 476.449,A -85,B 0,C 180,E1 -29706.902,E2 -29706.902} C_VEL
LIN {X 0,Y 127.771,Z 487.537,A -85,B 0,C 180,E1 -29708.086,E2 -29708.086} C_VEL
LIN {X 0,Y 117.588,Z 497.717,A -85,B 0,C 180,E1 -29709.549,E2 -29709.549} C_VEL
LIN {X 0,Y 105.839,Z 507.672,A -85,B 0,C 180,E1 -29711.666,E2 -29711.666} C_VEL
LIN {X 0,Y 95.984,Z 514.795,A -85,B 0,C 180,E1 -29714.035,E2 -29714.035} C_VEL
LIN {X 0,Y 84.612,Z 521.85,A -85,B 0,C 180,E1 -29717.218,E2 -29717.218} C_VEL
LIN {X 0,Y 72.025,Z 528.389,A -85,B 0,C 180,E1 -29722.034,E2 -29722.034} C_VEL
LIN {X 0,Y 60.167,Z 533.488,A -85,B 0,C 180,E1 -29728.832,E2 -29728.832} C_VEL
LIN {X 0,Y 52.006,Z 536.421,A -85,B 0,C 180,E1 -29735.825,E2 -29735.825} C_VEL
LIN {X 0,Y 42.716,Z 539.28,A -85,B 0,C 180,E1 -29748.844,E2 -29748.844} C_VEL
LIN {X 0,Y 36.405,Z 540.984,A -85,B 0,C 180,E1 -29767.289,E2 -29767.289} C_VEL
LIN {X 0,Y 34.328,Z 541.569,A -85,B 0,C 180,E1 -29790,E2 -29790} C_VEL
LIN {X 0,Y 36.397,Z 541.012,A -85,B 0,C 180,E1 -29812.717,E2 -29812.717} C_VEL
LIN {X 0,Y 42.668,Z 539.344,A -85,B 0,C 180,E1 -29831.212,E2 -29831.212} C_VEL
LIN {X 0,Y 51.99,Z 536.516,A -85,B 0,C 180,E1 -29844.199,E2 -29844.199} C_VEL
LIN {X 0,Y 63.045,Z 532.459,A -85,B 0,C 180,E1 -29853.099,E2 -29853.099} C_VEL
LIN {X 0,Y 75.099,Z 527.073,A -85,B 0,C 180,E1 -29859.358,E2 -29859.358} C_VEL
LIN {X 0,Y 87.783,Z 520.202,A -85,B 0,C 180,E1 -29863.886,E2 -29863.886} C_VEL
LIN {X 0,Y 99.237,Z 512.813,A -85,B 0,C 180,E1 -29866.844,E2 -29866.844} C_VEL
LIN {X 0,Y 109.158,Z 505.251,A -85,B 0,C 180,E1 -29869.061,E2 -29869.061} C_VEL
LIN {X 0,Y 119.265,Z 496.426,A -85,B 0,C 180,E1 -29870.755,E2 -29870.755} C_VEL
LIN {X 0,Y 129.442,Z 486.017,A -85,B 0,C 180,E1 -29872.243,E2 -29872.243} C_VEL
LIN {X 0,Y 138.846,Z 474.686,A -85,B 0,C 180,E1 -29873.384,E2 -29873.384} C_VEL
LIN {X 0,Y 147.763,Z 461.814,A -85,B 0,C 180,E1 -29874.392,E2 -29874.392} C_VEL
LIN {X 0,Y 155.161,Z 448.901,A -85,B 0,C 180,E1 -29875.179,E2 -29875.179} C_VEL
LIN {X 0,Y 161.637,Z 434.923,A -85,B 0,C 180,E1 -29875.789,E2 -29875.789} C_VEL
LIN {X 0,Y 167.221,Z 419.294,A -85,B 0,C 180,E1 -29876.277,E2 -29876.277} C_VEL
LIN {X 0,Y 171.021,Z 404.655,A -85,B 0,C 180,E1 -29876.614,E2 -29876.614} C_VEL
LIN {X 0,Y 172.821,Z 394.686,A -85,B 0,C 180,E1 -29876.809,E2 -29876.809} C_VEL
LIN {X 0,Y 172.824,Z 393.089,A -85,B 0,C 180,E1 -29879.417,E2 -29879.417} C_VEL
LIN {X 0,Y 172.812,Z 393.195,A -85,B 0,C 180,E1 -29880.291,E2 -29880.291} C_VEL
LIN {X 0,Y 172.835,Z 394.719,A -85,B 0,C 180,E1 -29882.879,E2 -29882.879} C_VEL
LIN {X 0,Y 170.094,Z 408.85,A -85,B 0,C 180,E1 -29883.108,E2 -29883.108} C_VEL
LIN {X 0,Y 165.665,Z 424.374,A -85,B 0,C 180,E1 -29883.422,E2 -29883.422} C_VEL
LIN {X 0,Y 160.236,Z 438.525,A -85,B 0,C 180,E1 -29883.804,E2 -29883.804} C_VEL
LIN {X 0,Y 153.285,Z 452.753,A -85,B 0,C 180,E1 -29884.29,E2 -29884.29} C_VEL
LIN {X 0,Y 145.495,Z 465.724,A -85,B 0,C 180,E1 -29884.965,E2 -29884.965} C_VEL
LIN {X 0,Y 137.457,Z 476.992,A -85,B 0,C 180,E1 -29885.794,E2 -29885.794} C_VEL
LIN {X 0,Y 127.434,Z 488.823,A -85,B 0,C 180,E1 -29886.938,E2 -29886.938} C_VEL
LIN {X 0,Y 117.173,Z 499.055,A -85,B 0,C 180,E1 -29888.255,E2 -29888.255} C_VEL
LIN {X 0,Y 105.343,Z 509.059,A -85,B 0,C 180,E1 -29890.255,E2 -29890.255} C_VEL
LIN {X 0,Y 93.673,Z 517.375,A -85,B 0,C 180,E1 -29892.753,E2 -29892.753} C_VEL
LIN {X 0,Y 80.686,Z 525.199,A -85,B 0,C 180,E1 -29896.642,E2 -29896.642} C_VEL
LIN {X 0,Y 68.125,Z 531.426,A -85,B 0,C 180,E1 -29901.807,E2 -29901.807} C_VEL
LIN {X 0,Y 56.393,Z 536.254,A -85,B 0,C 180,E1 -29909.266,E2 -29909.266} C_VEL
LIN {X 0,Y 46.035,Z 539.8,A -85,B 0,C 180,E1 -29920.243,E2 -29920.243} C_VEL
LIN {X 0,Y 38.113,Z 542.145,A -85,B 0,C 180,E1 -29936.414,E2 -29936.414} C_VEL
LIN {X 0,Y 34.255,Z 543.34,A -85,B 0,C 180,E1 -29958.161,E2 -29958.161} C_VEL
LIN {X 0,Y 34.142,Z 543.506,A -85,B 0,C 180,E1 -29970,E2 -29970} C_VEL
LIN {X 0,Y 35.603,Z 542.862,A -85,B 0,C 180,E1 -29993.253,E2 -29993.253} C_VEL
LIN {X 0,Y 41.662,Z 541.063,A -85,B 0,C 180,E1 -30012.434,E2 -30012.434} C_VEL
LIN {X 0,Y 50.944,Z 538.097,A -85,B 0,C 180,E1 -30025.864,E2 -30025.864} C_VEL
LIN {X 0,Y 62.121,Z 533.898,A -85,B 0,C 180,E1 -30034.831,E2 -30034.831} C_VEL
LIN {X 0,Y 74.318,Z 528.352,A -85,B 0,C 180,E1 -30041.023,E2 -30041.023} C_VEL
LIN {X 0,Y 87.131,Z 521.311,A -85,B 0,C 180,E1 -30045.442,E2 -30045.442} C_VEL
LIN {X 0,Y 98.644,Z 513.789,A -85,B 0,C 180,E1 -30048.41,E2 -30048.41} C_VEL
LIN {X 0,Y 110.398,Z 504.732,A -85,B 0,C 180,E1 -30050.651,E2 -30050.651} C_VEL
LIN {X 0,Y 120.587,Z 495.49,A -85,B 0,C 180,E1 -30052.208,E2 -30052.208} C_VEL
LIN {X 0,Y 130.86,Z 484.608,A -85,B 0,C 180,E1 -30053.486,E2 -30053.486} C_VEL
LIN {X 0,Y 140.317,Z 472.721,A -85,B 0,C 180,E1 -30054.55,E2 -30054.55} C_VEL
LIN {X 0,Y 148.953,Z 459.735,A -85,B 0,C 180,E1 -30055.349,E2 -30055.349} C_VEL
LIN {X 0,Y 156.752,Z 445.372,A -85,B 0,C 180,E1 -30055.995,E2 -30055.995} C_VEL
LIN {X 0,Y 162.602,Z 431.948,A -85,B 0,C 180,E1 -30056.394,E2 -30056.394} C_VEL
LIN {X 0,Y 167.833,Z 416.309,A -85,B 0,C 180,E1 -30056.741,E2 -30056.741} C_VEL
LIN {X 0,Y 171.53,Z 400.522,A -85,B 0,C 180,E1 -30056.988,E2 -30056.988} C_VEL
LIN {X 0,Y 172.541,Z 394.461,A -85,B 0,C 180,E1 -30057.115,E2 -30057.115} C_VEL
LIN {X 0,Y 172.545,Z 392.67,A -85,B 0,C 180,E1 -30060,E2 -30060} C_VEL
LIN {X 0,Y 172.491,Z 394.051,A -85,B 0,C 180,E1 -30062.644,E2 -30062.644} C_VEL
LIN {X 0,Y 172.515,Z 394.35,A -85,B 0,C 180,E1 -30063.133,E2 -30063.133} C_VEL
LIN {X 0,Y 172.462,Z 395.313,A -85,B 0,C 180,E1 -30063.62,E2 -30063.62} C_VEL
LIN {X 0,Y 172.121,Z 397.727,A -85,B 0,C 180,E1 -30063.966,E2 -30063.966} C_VEL
LIN {X 0,Y 171.472,Z 401.117,A -85,B 0,C 180,E1 -30063.945,E2 -30063.945} C_VEL
LIN {X 0,Y 170.261,Z 406.425,A -85,B 0,C 180,E1 -30063.415,E2 -30063.415} C_VEL
LIN {X 0,Y 167.149,Z 417.642,A -85,B 0,C 180,E1 -30061.817,E2 -30061.817} C_VEL
LIN {X 0,Y 165.684,Z 422.258,A -85,B 0,C 180,E1 -30061.506,E2 -30061.506} C_VEL
LIN {X 0,Y 164.886,Z 424.591,A -85,B 0,C 180,E1 -30061.515,E2 -30061.515} C_VEL
LIN {X 0,Y 159.095,Z 439.295,A -85,B 0,C 180,E1 -30061.927,E2 -30061.927} C_VEL
LIN {X 0,Y 152.183,Z 453.099,A -85,B 0,C 180,E1 -30062.471,E2 -30062.471} C_VEL
LIN {X 0,Y 144.299,Z 465.943,A -85,B 0,C 180,E1 -30063.222,E2 -30063.222} C_VEL
LIN {X 0,Y 134.753,Z 478.783,A -85,B 0,C 180,E1 -30064.106,E2 -30064.106} C_VEL
LIN {X 0,Y 125.239,Z 489.515,A -85,B 0,C 180,E1 -30065.095,E2 -30065.095} C_VEL
LIN {X 0,Y 114.902,Z 499.439,A -85,B 0,C 180,E1 -30066.325,E2 -30066.325} C_VEL
LIN {X 0,Y 104.103,Z 508.281,A -85,B 0,C 180,E1 -30067.921,E2 -30067.921} C_VEL
LIN {X 0,Y 94.513,Z 514.998,A -85,B 0,C 180,E1 -30069.855,E2 -30069.855} C_VEL
LIN {X 0,Y 82.779,Z 522.053,A -85,B 0,C 180,E1 -30072.49,E2 -30072.49} C_VEL
LIN {X 0,Y 69.669,Z 528.591,A -85,B 0,C 180,E1 -30076.602,E2 -30076.602} C_VEL
LIN {X 0,Y 57.07,Z 533.691,A -85,B 0,C 180,E1 -30082.545,E2 -30082.545} C_VEL
LIN {X 0,Y 48.177,Z 536.624,A -85,B 0,C 180,E1 -30088.926,E2 -30088.926} C_VEL
LIN {X 0,Y 37.638,Z 539.482,A -85,B 0,C 180,E1 -30101.678,E2 -30101.678} C_VEL
LIN {X 0,Y 29.962,Z 541.186,A -85,B 0,C 180,E1 -30122.023,E2 -30122.023} C_VEL
LIN {X 0,Y 27.245,Z 541.769,A -85,B 0,C 180,E1 -30150,E2 -30150} C_VEL
LIN {X 0,Y 29.954,Z 541.213,A -85,B 0,C 180,E1 -30177.985,E2 -30177.985} C_VEL
LIN {X 0,Y 37.599,Z 539.546,A -85,B 0,C 180,E1 -30198.387,E2 -30198.387} C_VEL
LIN {X 0,Y 48.165,Z 536.717,A -85,B 0,C 180,E1 -30211.101,E2 -30211.101} C_VEL
LIN {X 0,Y 61.738,Z 532.031,A -85,B 0,C 180,E1 -30220.031,E2 -30220.031} C_VEL
LIN {X 0,Y 72.893,Z 527.273,A -85,B 0,C 180,E1 -30224.606,E2 -30224.606} C_VEL
LIN {X 0,Y 86.073,Z 520.403,A -85,B 0,C 180,E1 -30228.462,E2 -30228.462} C_VEL
LIN {X 0,Y 97.857,Z 513.013,A -85,B 0,C 180,E1 -30230.925,E2 -30230.925} C_VEL
LIN {X 0,Y 108.033,Z 505.45,A -85,B 0,C 180,E1 -30232.773,E2 -30232.773} C_VEL
LIN {X 0,Y 118.333,Z 496.624,A -85,B 0,C 180,E1 -30234.147,E2 -30234.147} C_VEL
LIN {X 0,Y 128.677,Z 486.215,A -85,B 0,C 180,E1 -30235.373,E2 -30235.373} C_VEL
LIN {X 0,Y 138.208,Z 474.883,A -85,B 0,C 180,E1 -30236.306,E2 -30236.306} C_VEL
LIN {X 0,Y 146.867,Z 462.611,A -85,B 0,C 180,E1 -30237.107,E2 -30237.107} C_VEL
LIN {X 0,Y 154.727,Z 449.096,A -85,B 0,C 180,E1 -30237.795,E2 -30237.795} C_VEL
LIN {X 0,Y 161.272,Z 435.117,A -85,B 0,C 180,E1 -30238.296,E2 -30238.296} C_VEL
LIN {X 0,Y 166.935,Z 419.399,A -85,B 0,C 180,E1 -30238.716,E2 -30238.716} C_VEL
LIN {X 0,Y 170.766,Z 404.762,A -85,B 0,C 180,E1 -30238.987,E2 -30238.987} C_VEL
LIN {X 0,Y 171.598,Z 400.456,A -85,B 0,C 180,E1 -30239.091,E2 -30239.091} C_VEL
LIN {X 0,Y 171.631,Z 400.264,A -85,B 0,C 180,E1 -30240.175,E2 -30240.175} C_VEL
LIN {X 0,Y 171.595,Z 400.525,A -85,B 0,C 180,E1 -30240.591,E2 -30240.591} C_VEL
LIN {X 0,Y 168.106,Z 415.42,A -85,B 0,C 180,E1 -30240.821,E2 -30240.821} C_VEL
LIN {X 0,Y 163.423,Z 429.734,A -85,B 0,C 180,E1 -30241.087,E2 -30241.087} C_VEL
LIN {X 0,Y 157.294,Z 444.08,A -85,B 0,C 180,E1 -30241.386,E2 -30241.386} C_VEL
LIN {X 0,Y 150.294,Z 457.213,A -85,B 0,C 180,E1 -30241.804,E2 -30241.804} C_VEL
LIN {X 0,Y 141.561,Z 470.603,A -85,B 0,C 180,E1 -30242.414,E2 -30242.414} C_VEL
LIN {X 0,Y 131.985,Z 482.81,A -85,B 0,C 180,E1 -30243.257,E2 -30243.257} C_VEL
LIN {X 0,Y 121.564,Z 493.959,A -85,B 0,C 180,E1 -30244.25,E2 -30244.25} C_VEL
LIN {X 0,Y 111.185,Z 503.348,A -85,B 0,C 180,E1 -30245.418,E2 -30245.418} C_VEL
LIN {X 0,Y 99.168,Z 512.589,A -85,B 0,C 180,E1 -30247.184,E2 -30247.184} C_VEL
LIN {X 0,Y 87.718,Z 520.022,A -85,B 0,C 180,E1 -30249.394,E2 -30249.394} C_VEL
LIN {X 0,Y 75.618,Z 526.671,A -85,B 0,C 180,E1 -30252.615,E2 -30252.615} C_VEL
LIN {X 0,Y 62.593,Z 532.547,A -85,B 0,C 180,E1 -30257.375,E2 -30257.375} C_VEL
LIN {X 0,Y 49.332,Z 537.348,A -85,B 0,C 180,E1 -30265.301,E2 -30265.301} C_VEL
LIN {X 0,Y 36.709,Z 540.917,A -85,B 0,C 180,E1 -30280.023,E2 -30280.023} C_VEL
LIN {X 0,Y 29.174,Z 542.683,A -85,B 0,C 180,E1 -30301.198,E2 -30301.198} C_VEL
LIN {X 0,Y 27.028,Z 543.305,A -85,B 0,C 180,E1 -30330,E2 -30330} C_VEL
LIN {X 0,Y 29.156,Z 542.659,A -85,B 0,C 180,E1 -30358.822,E2 -30358.822} C_VEL
LIN {X 0,Y 36.691,Z 540.86,A -85,B 0,C 180,E1 -30380.012,E2 -30380.012} C_VEL
LIN {X 0,Y 48.951,Z 537.373,A -85,B 0,C 180,E1 -30394.488,E2 -30394.488} C_VEL
LIN {X 0,Y 62.586,Z 532.436,A -85,B 0,C 180,E1 -30402.646,E2 -30402.646} C_VEL
LIN {X 0,Y 75.612,Z 526.52,A -85,B 0,C 180,E1 -30407.403,E2 -30407.403} C_VEL
LIN {X 0,Y 89.968,Z 518.471,A -85,B 0,C 180,E1 -30411.115,E2 -30411.115} C_VEL
LIN {X 0,Y 102.593,Z 509.881,A -85,B 0,C 180,E1 -30413.356,E2 -30413.356} C_VEL
LIN {X 0,Y 114.634,Z 500.086,A -85,B 0,C 180,E1 -30415.025,E2 -30415.025} C_VEL
LIN {X 0,Y 125.035,Z 490.079,A -85,B 0,C 180,E1 -30416.09,E2 -30416.09} C_VEL
LIN {X 0,Y 135.287,Z 478.407,A -85,B 0,C 180,E1 -30417.06,E2 -30417.06} C_VEL
LIN {X 0,Y 144.177,Z 466.337,A -85,B 0,C 180,E1 -30417.796,E2 -30417.796} C_VEL
LIN {X 0,Y 152.044,Z 453.536,A -85,B 0,C 180,E1 -30418.299,E2 -30418.299} C_VEL
LIN {X 0,Y 158.169,Z 441.543,A -85,B 0,C 180,E1 -30418.669,E2 -30418.669} C_VEL
LIN {X 0,Y 164.201,Z 426.738,A -85,B 0,C 180,E1 -30418.987,E2 -30418.987} C_VEL
LIN {X 0,Y 168.684,Z 412.18,A -85,B 0,C 180,E1 -30419.212,E2 -30419.212} C_VEL
LIN {X 0,Y 171.322,Z 400.201,A -85,B 0,C 180,E1 -30419.415,E2 -30419.415} C_VEL
LIN {X 0,Y 171.373,Z 399.834,A -85,B 0,C 180,E1 -30420,E2 -30420} C_VEL
LIN {X 0,Y 171.313,Z 400.194,A -85,B 0,C 180,E1 -30421.015,E2 -30421.015} C_VEL
LIN {X 0,Y 167.803,Z 415.226,A -85,B 0,C 180,E1 -30421.301,E2 -30421.301} C_VEL
LIN {X 0,Y 164.886,Z 424.591,A -85,B 0,C 180,E1 -30421.515,E2 -30421.515} C_VEL
LIN {X 0,Y 164.78,Z 425.242,A -85,B 0,C 180,E1 -30421.523,E2 -30421.523} C_VEL
LIN {X 0,Y 164.78,Z 482.984,A -85,B 0,C 180,E1 -30421.523,E2 -30421.523} C_VEL
LIN {X 0,Y 146.085,Z 482.984,A -85,B 0,C 180,E1 -30420.53,E2 -30420.53} C_VEL
LIN {X 0,Y 144.108,Z 480.984,A -85,B 0,C 180,E1 -30420.409,E2 -30420.409} C_VEL
LIN {X 0,Y 144.108,Z 472.335,A -85,B 0,C 180,E1 -30420.409,E2 -30420.409} C_VEL
LIN {X 0,Y 140.566,Z 471.124,A -85,B 0,C 180,E1 -30420.648,E2 -30420.648} C_VEL
LIN {X 0,Y 131.144,Z 482.881,A -85,B 0,C 180,E1 -30421.333,E2 -30421.333} C_VEL
LIN {X 0,Y 121.318,Z 493.255,A -85,B 0,C 180,E1 -30422.175,E2 -30422.175} C_VEL
LIN {X 0,Y 110.855,Z 502.597,A -85,B 0,C 180,E1 -30423.141,E2 -30423.141} C_VEL
LIN {X 0,Y 100.712,Z 510.364,A -85,B 0,C 180,E1 -30424.41,E2 -30424.41} C_VEL
LIN {X 0,Y 90.104,Z 517.394,A -85,B 0,C 180,E1 -30426.034,E2 -30426.034} C_VEL
LIN {X 0,Y 78.127,Z 524.051,A -85,B 0,C 180,E1 -30428.314,E2 -30428.314} C_VEL
LIN {X 0,Y 64.626,Z 530.204,A -85,B 0,C 180,E1 -30431.843,E2 -30431.843} C_VEL
LIN {X 0,Y 51.493,Z 534.944,A -85,B 0,C 180,E1 -30437.181,E2 -30437.181} C_VEL
LIN {X 0,Y 39.034,Z 538.405,A -85,B 0,C 180,E1 -30445.813,E2 -30445.813} C_VEL
LIN {X 0,Y 28.177,Z 540.676,A -85,B 0,C 180,E1 -30461.561,E2 -30461.561} C_VEL
LIN {X 0,Y 21.082,Z 541.821,A -85,B 0,C 180,E1 -30490.527,E2 -30490.527} C_VEL
LIN {X 0,Y 20.156,Z 541.97,A -85,B 0,C 180,E1 -30510,E2 -30510} C_VEL
LIN {X 0,Y 23.909,Z 541.414,A -85,B 0,C 180,E1 -30546.007,E2 -30546.007} C_VEL
LIN {X 0,Y 33.285,Z 539.747,A -85,B 0,C 180,E1 -30567.625,E2 -30567.625} C_VEL
LIN {X 0,Y 45.152,Z 536.918,A -85,B 0,C 180,E1 -30579.05,E2 -30579.05} C_VEL
LIN {X 0,Y 58.952,Z 532.503,A -85,B 0,C 180,E1 -30586.205,E2 -30586.205} C_VEL
LIN {X 0,Y 71.331,Z 527.474,A -85,B 0,C 180,E1 -30590.142,E2 -30590.142} C_VEL
LIN {X 0,Y 84.934,Z 520.603,A -85,B 0,C 180,E1 -30593.186,E2 -30593.186} C_VEL
LIN {X 0,Y 96.988,Z 513.213,A -85,B 0,C 180,E1 -30595.092,E2 -30595.092} C_VEL
LIN {X 0,Y 105.632,Z 506.996,A -85,B 0,C 180,E1 -30596.345,E2 -30596.345} C_VEL
LIN {X 0,Y 116.076,Z 498.439,A -85,B 0,C 180,E1 -30597.432,E2 -30597.432} C_VEL
LIN {X 0,Y 126.55,Z 488.295,A -85,B 0,C 180,E1 -30598.398,E2 -30598.398} C_VEL
